	LOCAL CONST Robtarget Tr_meulage_bavure_P139 :=[[-127.011234375,174.2020625,18.5],[0.190442175287024,-0.303310117531916,0.790723364420333,-0.496478913383551],[0,0,0,0],[8.999999E+09,8.999999E+09,8.999999E+09,8.999999E+09,8.999999E+09,8.999999E+09]];
	LOCAL CONST Robtarget Tr_meulage_bavure_P140 :=[[-124.162203125,176.750703125,18.5],[0.192518086359884,-0.306201340616146,0.789260106907647,-0.496231809816071],[0,0,0,0],[8.999999E+09,8.999999E+09,8.999999E+09,8.999999E+09,8.999999E+09,8.999999E+09]];
	LOCAL CONST Robtarget Tr_meulage_bavure_P141 :=[[-122.8513828125,177.964453125,18.5],[0.194663155240253,-0.309123590669608,0.787712135243574,-0.49604279419567],[0,0,0,0],[8.999999E+09,8.999999E+09,8.999999E+09,8.999999E+09,8.999999E+09,8.999999E+09]];
	LOCAL CONST Robtarget Tr_meulage_bavure_P142 :=[[-119.9177578125,180.693,18.5],[0.196899901424474,-0.312103049014616,0.786062139961331,-0.495911713648938],[0,0,0,0],[8.999999E+09,8.999999E+09,8.999999E+09,8.999999E+09,8.999999E+09,8.999999E+09]];
	LOCAL CONST Robtarget Tr_meulage_bavure_P143 :=[[-116.7352265625,183.69171875,18.5],[0.199318008553782,-0.315263950024278,0.784246523173782,-0.49582089928832],[0,0,0,0],[8.999999E+09,8.999999E+09,8.999999E+09,8.999999E+09,8.999999E+09,8.999999E+09]];
	LOCAL CONST Robtarget Tr_meulage_bavure_P144 :=[[-116.454375,183.9246875,18.5],[0.20211682598174,-0.318902881092808,0.782129693912803,-0.495704431073234],[0,0,0,0],[8.999999E+09,8.999999E+09,8.999999E+09,8.999999E+09,8.999999E+09,8.999999E+09]];
	LOCAL CONST Robtarget Tr_meulage_bavure_P145 :=[[-112.0714453125,188.2565625,18.5],[0.205596230982278,-0.323472429632436,0.779505217686998,-0.495446659765022],[0,0,0,0],[8.999999E+09,8.999999E+09,8.999999E+09,8.999999E+09,8.999999E+09,8.999999E+09]];
	LOCAL CONST Robtarget Tr_meulage_bavure_P146 :=[[-110.354734375,189.926171875,18.5],[0.210070493146241,-0.329436360615377,0.776142089251371,-0.494919720264112],[0,0,0,0],[8.999999E+09,8.999999E+09,8.999999E+09,8.999999E+09,8.999999E+09,8.999999E+09]];
	LOCAL CONST Robtarget Tr_meulage_bavure_P147 :=[[-106.4182109375,193.63390625,18.5],[0.215682425483319,-0.33696654676811,0.771899664135642,-0.494070385880484],[0,0,0,0],[8.999999E+09,8.999999E+09,8.999999E+09,8.999999E+09,8.999999E+09,8.999999E+09]];
	LOCAL CONST Robtarget Tr_meulage_bavure_P148 :=[[-103.6989765625,196.126,18.5],[0.222270904527529,-0.345759095574698,0.766835763229423,-0.492959638368325],[0,0,0,0],[8.999999E+09,8.999999E+09,8.999999E+09,8.999999E+09,8.999999E+09,8.999999E+09]];
	LOCAL CONST Robtarget Tr_meulage_bavure_P149 :=[[-101.426390625,198.445984375,18.5],[0.229322634138018,-0.354960138136149,0.761267985475532,-0.491818547938559],[0,0,0,0],[8.999999E+09,8.999999E+09,8.999999E+09,8.999999E+09,8.999999E+09,8.999999E+09]];
	LOCAL CONST Robtarget Tr_meulage_bavure_P150 :=[[-101.17571875,198.708734375,18.5],[0.236006383142285,-0.363228319091028,0.755788103274612,-0.491070787437991],[0,0,0,0],[8.999999E+09,8.999999E+09,8.999999E+09,8.999999E+09,8.999999E+09,8.999999E+09]];
	LOCAL CONST Robtarget Tr_meulage_bavure_P151 :=[[-100.905703125,199.091640625,18.5],[0.241370828071747,-0.36906936863497,0.751137903082245,-0.491243091599823],[0,0,0,0],[8.999999E+09,8.999999E+09,8.999999E+09,8.999999E+09,8.999999E+09,8.999999E+09]];
	LOCAL CONST Robtarget Tr_meulage_bavure_P152 :=[[-99.122953125,201.35684375,18.5],[0.244403323371577,-0.370940628519687,0.748128933610927,-0.492923081557889],[0,0,0,0],[8.999999E+09,8.999999E+09,8.999999E+09,8.999999E+09,8.999999E+09,8.999999E+09]];
	LOCAL CONST Robtarget Tr_meulage_bavure_P153 :=[[-96.8828125,205.6408125,18.5],[0.244018753605267,-0.367253165730394,0.747565690475479,-0.496714705413334],[0,0,0,0],[8.999999E+09,8.999999E+09,8.999999E+09,8.999999E+09,8.999999E+09,8.999999E+09]];
	LOCAL CONST Robtarget Tr_meulage_bavure_P154 :=[[-96.362,206.638734375,18.5],[0.239111744899531,-0.356478263353551,0.750077508931146,-0.50312279992382],[0,0,0,0],[8.999999E+09,8.999999E+09,8.999999E+09,8.999999E+09,8.999999E+09,8.999999E+09]];
	LOCAL CONST Robtarget Tr_meulage_bavure_P155 :=[[-95.8127421875,207.699921875,18.5],[0.228678070464608,-0.337329813828571,0.755875580230949,-0.512412962366772],[0,0,0,0],[8.999999E+09,8.999999E+09,8.999999E+09,8.999999E+09,8.999999E+09,8.999999E+09]];
	LOCAL CONST Robtarget Tr_meulage_bavure_P156 :=[[-94.308015625,209.90903125,18.5],[0.212075421526648,-0.309184782305918,0.764495371744153,-0.524381171054517],[0,0,0,0],[8.999999E+09,8.999999E+09,8.999999E+09,8.999999E+09,8.999999E+09,8.999999E+09]];
	LOCAL CONST Robtarget Tr_meulage_bavure_P157 :=[[-93.75003125,210.7380625,18.5],[0.189378915500843,-0.272552593388089,0.774672329708009,-0.538268977172116],[0,0,0,0],[8.999999E+09,8.999999E+09,8.999999E+09,8.999999E+09,8.999999E+09,8.999999E+09]];
	LOCAL CONST Robtarget Tr_meulage_bavure_P158 :=[[-91.9986875,212.56409375,18.5],[0.161390602222789,-0.22902506301056,0.784689128838321,-0.552958918103443],[0,0,0,0],[8.999999E+09,8.999999E+09,8.999999E+09,8.999999E+09,8.999999E+09,8.999999E+09]];
	LOCAL CONST Robtarget Tr_meulage_bavure_P159 :=[[-91.4162265625,213.00103125,18.5],[0.129000654455637,-0.180301065959294,0.793038362347405,-0.567398019567663],[0,0,0,0],[8.999999E+09,8.999999E+09,8.999999E+09,8.999999E+09,8.999999E+09,8.999999E+09]];
	LOCAL CONST Robtarget Tr_meulage_bavure_P160 :=[[-91.3440546875,213.013484375,18.5],[0.0922817945694316,-0.126902080153844,0.798750290191089,-0.580842410954403],[0,0,0,0],[8.999999E+09,8.999999E+09,8.999999E+09,8.999999E+09,8.999999E+09,8.999999E+09]];
	LOCAL CONST Robtarget Tr_meulage_bavure_P161 :=[[-89.162078125,213.66828125,18.5],[0.0503174553587556,-0.0680160169269533,0.801040840932036,-0.592600663420577],[0,0,0,0],[8.999999E+09,8.999999E+09,8.999999E+09,8.999999E+09,8.999999E+09,8.999999E+09]];
	LOCAL CONST Robtarget Tr_meulage_bavure_P162 :=[[-88.3440546875,213.92571875,18.5],[0.00252406567631668,-0.00335106739002913,0.798759606326067,-0.601635679412081],[0,0,0,0],[8.999999E+09,8.999999E+09,8.999999E+09,8.999999E+09,8.999999E+09,8.999999E+09]];
	LOCAL CONST Robtarget Tr_meulage_bavure_P163 :=[[-87.4652109375,213.682671875,18.5],[0.0493797498258951,-0.0643494973435124,-0.79072352084382,0.606775985090975],[0,0,0,0],[8.999999E+09,8.999999E+09,8.999999E+09,8.999999E+09,8.999999E+09,8.999999E+09]];
	LOCAL CONST Robtarget Tr_meulage_bavure_P164 :=[[-85.52471875,212.9560625,18.5],[0.100577948139047,-0.128593194746078,-0.777116334377217,0.607814173458676],[0,0,0,0],[8.999999E+09,8.999999E+09,8.999999E+09,8.999999E+09,8.999999E+09,8.999999E+09]];
	LOCAL CONST Robtarget Tr_meulage_bavure_P165 :=[[-84.909671875,212.780703125,18.5],[0.145497398822093,-0.182465256610375,-0.760270957778014,0.606238408404991],[0,0,0,0],[8.999999E+09,8.999999E+09,8.999999E+09,8.999999E+09,8.999999E+09,8.999999E+09]];
	LOCAL CONST Robtarget Tr_meulage_bavure_P166 :=[[-84.38684375,212.302609375,18.5],[0.1809439145775,-0.222567903189488,-0.743324803089797,0.604310404807596],[0,0,0,0],[8.999999E+09,8.999999E+09,8.999999E+09,8.999999E+09,8.999999E+09,8.999999E+09]];
	LOCAL CONST Robtarget Tr_meulage_bavure_P167 :=[[-83.17071875,211.42740625,18.5],[0.206769871621223,-0.249506095485494,-0.728419709809437,0.603653588464826],[0,0,0,0],[8.999999E+09,8.999999E+09,8.999999E+09,8.999999E+09,8.999999E+09,8.999999E+09]];
	LOCAL CONST Robtarget Tr_meulage_bavure_P168 :=[[-80.6744375,209.227359375,18.5],[0.2245846611902,-0.265959685221285,-0.716250493467956,0.604824277292163],[0,0,0,0],[8.999999E+09,8.999999E+09,8.999999E+09,8.999999E+09,8.999999E+09,8.999999E+09]];
	LOCAL CONST Robtarget Tr_meulage_bavure_P169 :=[[-78.3284921875,206.867765625,18.5],[0.236502082156785,-0.27502158665567,-0.706570578623321,0.607608352010412],[0,0,0,0],[8.999999E+09,8.999999E+09,8.999999E+09,8.999999E+09,8.999999E+09,8.999999E+09]];
	LOCAL CONST Robtarget Tr_meulage_bavure_P170 :=[[-78.2308046875,206.771265625,18.5],[0.244452716764455,-0.279349107845849,-0.698778256751739,0.611486625449164],[0,0,0,0],[8.999999E+09,8.999999E+09,8.999999E+09,8.999999E+09,8.999999E+09,8.999999E+09]];
	LOCAL CONST Robtarget Tr_meulage_bavure_P171 :=[[-78.2126171875,206.752984375,18.5],[0.249940631640984,-0.280932693864888,-0.692284568560228,0.61591280089482],[0,0,0,0],[8.999999E+09,8.999999E+09,8.999999E+09,8.999999E+09,8.999999E+09,8.999999E+09]];
	LOCAL CONST Robtarget Tr_meulage_bavure_P172 :=[[-78.1261015625,206.67025,18.5],[0.253945556991537,-0.28103631183058,-0.686678755595343,0.620485722745459],[0,0,0,0],[8.999999E+09,8.999999E+09,8.999999E+09,8.999999E+09,8.999999E+09,8.999999E+09]];
	LOCAL CONST Robtarget Tr_meulage_bavure_P173 :=[[-71.4190078125,200.202265625,18.5],[0.256989223430704,-0.28033188921564,-0.681743993140734,0.62497655855704],[0,0,0,0],[8.999999E+09,8.999999E+09,8.999999E+09,8.999999E+09,8.999999E+09,8.999999E+09]];
	LOCAL CONST Robtarget Tr_meulage_bavure_P174 :=[[-69.085453125,198.020046875,18.5],[0.259270883175515,-0.279099527691383,-0.677410081478571,0.629283437165663],[0,0,0,0],[8.999999E+09,8.999999E+09,8.999999E+09,8.999999E+09,8.999999E+09,8.999999E+09]];
	LOCAL CONST Robtarget Tr_meulage_bavure_P175 :=[[-67.2452734375,196.310515625,18.5],[0.260735300009118,-0.277312443707638,-0.673704973181902,0.633432333405887],[0,0,0,0],[8.999999E+09,8.999999E+09,8.999999E+09,8.999999E+09,8.999999E+09,8.999999E+09]];
	LOCAL CONST Robtarget Tr_meulage_bavure_P176 :=[[-65.573640625,194.69784375,18.5],[0.261286645683991,-0.274898585018902,-0.670672090802852,0.63746294273467],[0,0,0,0],[8.999999E+09,8.999999E+09,8.999999E+09,8.999999E+09,8.999999E+09,8.999999E+09]];
	LOCAL CONST Robtarget Tr_meulage_bavure_P177 :=[[-61.1885078125,190.282375,18.5],[0.260938532941136,-0.27189092460859,-0.668297686772354,0.641377119171501],[0,0,0,0],[8.999999E+09,8.999999E+09,8.999999E+09,8.999999E+09,8.999999E+09,8.999999E+09]];
	LOCAL CONST Robtarget Tr_meulage_bavure_P178 :=[[-60.0119609375,189.182125,18.5],[0.259877003328182,-0.268486303796629,-0.666487105011264,0.645115483203196],[0,0,0,0],[8.999999E+09,8.999999E+09,8.999999E+09,8.999999E+09,8.999999E+09,8.999999E+09]];
	LOCAL CONST Robtarget Tr_meulage_bavure_P179 :=[[-56.05679296875,185.29428125,18.5],[0.258463269105114,-0.265048735721945,-0.665076369193805,0.648551716793412],[0,0,0,0],[8.999999E+09,8.999999E+09,8.999999E+09,8.999999E+09,8.999999E+09,8.999999E+09]];
	LOCAL CONST Robtarget Tr_meulage_bavure_P180 :=[[-54.05676171875,183.442875,18.5],[0.257127057998321,-0.26199711676235,-0.663881001079455,0.651540638225341],[0,0,0,0],[8.999999E+09,8.999999E+09,8.999999E+09,8.999999E+09,8.999999E+09,8.999999E+09]];
	LOCAL CONST Robtarget Tr_meulage_bavure_P181 :=[[-52.6292734375,182.20425,18.5],[0.25621924205441,-0.259657247241297,-0.662753509176958,0.653978287124094],[0,0,0,0],[8.999999E+09,8.999999E+09,8.999999E+09,8.999999E+09,8.999999E+09,8.999999E+09]];
	LOCAL CONST Robtarget Tr_meulage_bavure_P182 :=[[-50.96499609375,180.630546875,18.5],[0.25590306679538,-0.258163340391161,-0.661625616240868,0.655832946730102],[0,0,0,0],[8.999999E+09,8.999999E+09,8.999999E+09,8.999999E+09,8.999999E+09,8.999999E+09]];
	LOCAL CONST Robtarget Tr_meulage_bavure_P183 :=[[-48.427734375,178.2460625,18.5],[0.256144256103112,-0.257446199530212,-0.66049710199585,0.657156870669339],[0,0,0,0],[8.999999E+09,8.999999E+09,8.999999E+09,8.999999E+09,8.999999E+09,8.999999E+09]];
	LOCAL CONST Robtarget Tr_meulage_bavure_P184 :=[[-43.8993828125,173.85284375,18.5],[0.25677948279759,-0.257318314364314,-0.659420499348961,0.658039654842531],[0,0,0,0],[8.999999E+09,8.999999E+09,8.999999E+09,8.999999E+09,8.999999E+09,8.999999E+09]];
	LOCAL CONST Robtarget Tr_meulage_bavure_P185 :=[[-43.0797734375,173.100734375,18.5],[0.257617067745429,-0.257566704531451,-0.658453973298864,0.658582723862382],[0,0,0,0],[8.999999E+09,8.999999E+09,8.999999E+09,8.999999E+09,8.999999E+09,8.999999E+09]];
	LOCAL CONST Robtarget Tr_meulage_bavure_P186 :=[[-41.48028515625,171.667078125,18.5],[0.258515279559301,-0.258032413744623,-0.657635522171516,0.658866180396063],[0,0,0,0],[8.999999E+09,8.999999E+09,8.999999E+09,8.999999E+09,8.999999E+09,8.999999E+09]];
	LOCAL CONST Robtarget Tr_meulage_bavure_P187 :=[[-39.0978984375,169.191015625,18.5],[0.259401397972076,-0.258624835211619,-0.656973453033344,0.658946121736322],[0,0,0,0],[8.999999E+09,8.999999E+09,8.999999E+09,8.999999E+09,8.999999E+09,8.999999E+09]];
	LOCAL CONST Robtarget Tr_meulage_bavure_P188 :=[[-38.23126171875,168.3086875,18.5],[0.260254131673374,-0.259304274264351,-0.656454947464892,0.658859607385399],[0,0,0,0],[8.999999E+09,8.999999E+09,8.999999E+09,8.999999E+09,8.999999E+09,8.999999E+09]];
	LOCAL CONST Robtarget Tr_meulage_bavure_P189 :=[[-35.4189765625,165.67340625,18.5],[0.26105089862492,-0.260039320067026,-0.656077957241587,0.658630165091083],[0,0,0,0],[8.999999E+09,8.999999E+09,8.999999E+09,8.999999E+09,8.999999E+09,8.999999E+09]];
	LOCAL CONST Robtarget Tr_meulage_bavure_P190 :=[[-34.5329296875,164.8164375,18.5],[0.261759260875739,-0.2607857252386,-0.655841250825685,0.65828956286194],[0,0,0,0],[8.999999E+09,8.999999E+09,8.999999E+09,8.999999E+09,8.999999E+09,8.999999E+09]];
	LOCAL CONST Robtarget Tr_meulage_bavure_P191 :=[[-31.362640625,161.758390625,18.5],[0.262331145993118,-0.261476154519974,-0.655742298154861,0.657886486310493],[0,0,0,0],[8.999999E+09,8.999999E+09,8.999999E+09,8.999999E+09,8.999999E+09,8.999999E+09]];
	LOCAL CONST Robtarget Tr_meulage_bavure_P192 :=[[-30.35272265625,160.788,18.5],[0.262709953836354,-0.262042168547561,-0.655790615320609,0.657461824683083],[0,0,0,0],[8.999999E+09,8.999999E+09,8.999999E+09,8.999999E+09,8.999999E+09,8.999999E+09]];
	LOCAL CONST Robtarget Tr_meulage_bavure_P193 :=[[-30.05163671875,160.490046875,18.5],[0.262861381702475,-0.262436848617029,-0.655986833448376,0.657047995841857],[0,0,0,0],[8.999999E+09,8.999999E+09,8.999999E+09,8.999999E+09,8.999999E+09,8.999999E+09]];
	LOCAL CONST Robtarget Tr_meulage_bavure_P194 :=[[-28.3164375,158.80840625,18.5],[0.262783789530265,-0.262648406055636,-0.656321684574613,0.656659988969703],[0,0,0,0],[8.999999E+09,8.999999E+09,8.999999E+09,8.999999E+09,8.999999E+09,8.999999E+09]];
	LOCAL CONST Robtarget Tr_meulage_bavure_P195 :=[[-23.402556640625,154.107609375,18.5],[0.262525712244518,-0.262712755695221,-0.6567633663921,0.656295770953042],[0,0,0,0],[8.999999E+09,8.999999E+09,8.999999E+09,8.999999E+09,8.999999E+09,8.999999E+09]];
	LOCAL CONST Robtarget Tr_meulage_bavure_P196 :=[[-20.412109375,151.27234375,18.5],[0.262165502805967,-0.262695654197738,-0.657267884152523,0.655941438594775],[0,0,0,0],[8.999999E+09,8.999999E+09,8.999999E+09,8.999999E+09,8.999999E+09,8.999999E+09]];
	LOCAL CONST Robtarget Tr_meulage_bavure_P197 :=[[-16.22085546875,147.224703125,18.5],[0.261778886975614,-0.262664639311416,-0.657796488234147,0.655578280341895],[0,0,0,0],[8.999999E+09,8.999999E+09,8.999999E+09,8.999999E+09,8.999999E+09,8.999999E+09]];
	LOCAL CONST Robtarget Tr_meulage_bavure_P198 :=[[-14.92822265625,146.00884375,18.5],[0.261413667950097,-0.262658057795985,-0.658319979987044,0.655201070537568],[0,0,0,0],[8.999999E+09,8.999999E+09,8.999999E+09,8.999999E+09,8.999999E+09,8.999999E+09]];
	LOCAL CONST Robtarget Tr_meulage_bavure_P199 :=[[-11.3293759765625,142.66771875,18.5],[0.261077038101035,-0.262673384522033,-0.658825150616152,0.654821268863295],[0,0,0,0],[8.999999E+09,8.999999E+09,8.999999E+09,8.999999E+09,8.999999E+09,8.999999E+09]];
	LOCAL CONST Robtarget Tr_meulage_bavure_P200 :=[[-6.89715576171875,138.38053125,18.5],[0.260745670082175,-0.262685448847026,-0.659319494058335,0.654450804302429],[0,0,0,0],[8.999999E+09,8.999999E+09,8.999999E+09,8.999999E+09,8.999999E+09,8.999999E+09]];
	LOCAL CONST Robtarget Tr_meulage_bavure_P201 :=[[-5.350982421875,136.87134375,18.5],[0.260409251060274,-0.262675169776875,-0.659798086716118,0.654106460685619],[0,0,0,0],[8.999999E+09,8.999999E+09,8.999999E+09,8.999999E+09,8.999999E+09,8.999999E+09]];
	LOCAL CONST Robtarget Tr_meulage_bavure_P202 :=[[-2.4296875,134.151703125,18.5],[0.260088169520179,-0.262658023455088,-0.660247459881271,0.653787579042795],[0,0,0,0],[8.999999E+09,8.999999E+09,8.999999E+09,8.999999E+09,8.999999E+09,8.999999E+09]];
	LOCAL CONST Robtarget Tr_meulage_bavure_P203 :=[[0.08966064453125,131.796015625,18.5],[0.259835082530743,-0.2626829624302,-0.660641959735919,0.653479603485389],[0,0,0,0],[8.999999E+09,8.999999E+09,8.999999E+09,8.999999E+09,8.999999E+09,8.999999E+09]];
	LOCAL CONST Robtarget Tr_meulage_bavure_P204 :=[[10.1913759765625,122.3306875,18.5],[0.259705705094535,-0.262804592862917,-0.660957113707128,0.653163368960209],[0,0,0,0],[8.999999E+09,8.999999E+09,8.999999E+09,8.999999E+09,8.999999E+09,8.999999E+09]];
	LOCAL CONST Robtarget Tr_meulage_bavure_P205 :=[[11.085693359375,121.4689921875,18.5],[0.259721319569318,-0.263044848045246,-0.661184340698121,0.652830385087595],[0,0,0,0],[8.999999E+09,8.999999E+09,8.999999E+09,8.999999E+09,8.999999E+09,8.999999E+09]];
	LOCAL CONST Robtarget Tr_meulage_bavure_P206 :=[[17.055603515625,115.9521796875,18.5],[0.259852146003557,-0.263371187191271,-0.661332752660767,0.652496337332969],[0,0,0,0],[8.999999E+09,8.999999E+09,8.999999E+09,8.999999E+09,8.999999E+09,8.999999E+09]];
	LOCAL CONST Robtarget Tr_meulage_bavure_P207 :=[[21.760802734375,111.515078125,18.5],[0.260013158425684,-0.263699039363099,-0.661438173618062,0.652192852280122],[0,0,0,0],[8.999999E+09,8.999999E+09,8.999999E+09,8.999999E+09,8.999999E+09,8.999999E+09]];
	LOCAL CONST Robtarget Tr_meulage_bavure_P208 :=[[27.258392578125,106.207,18.5],[0.260100750372149,-0.263922045498253,-0.661541379549992,0.651963002553792],[0,0,0,0],[8.999999E+09,8.999999E+09,8.999999E+09,8.999999E+09,8.999999E+09,8.999999E+09]];
	LOCAL CONST Robtarget Tr_meulage_bavure_P209 :=[[28.722015625,104.805484375,18.5],[0.260029172084293,-0.263956096433542,-0.661680511567474,0.651836566504618],[0,0,0,0],[8.999999E+09,8.999999E+09,8.999999E+09,8.999999E+09,8.999999E+09,8.999999E+09]];
	LOCAL CONST Robtarget Tr_meulage_bavure_P210 :=[[29.41101171875,104.1642734375,18.5],[0.259754440439883,-0.263762334346421,-0.661879667905148,0.651822343024279],[0,0,0,0],[8.999999E+09,8.999999E+09,8.999999E+09,8.999999E+09,8.999999E+09,8.999999E+09]];
	LOCAL CONST Robtarget Tr_meulage_bavure_P211 :=[[32.655669921875,101.1337265625,18.5],[0.259303936814273,-0.263365032759278,-0.662124089734479,0.651914118320513],[0,0,0,0],[8.999999E+09,8.999999E+09,8.999999E+09,8.999999E+09,8.999999E+09,8.999999E+09]];
	LOCAL CONST Robtarget Tr_meulage_bavure_P212 :=[[33.78524609375,100.0587734375,18.5],[0.258758312179959,-0.262849754312713,-0.662384650536248,0.65207416546701],[0,0,0,0],[8.999999E+09,8.999999E+09,8.999999E+09,8.999999E+09,8.999999E+09,8.999999E+09]];
	LOCAL CONST Robtarget Tr_meulage_bavure_P213 :=[[36.34820703125,97.613921875,18.5],[0.258230341869406,-0.262336593473032,-0.662621353895246,0.652249602242122],[0,0,0,0],[8.999999E+09,8.999999E+09,8.999999E+09,8.999999E+09,8.999999E+09,8.999999E+09]];
	LOCAL CONST Robtarget Tr_meulage_bavure_P214 :=[[36.68661328125,97.301265625,18.5],[0.257838264135803,-0.261942230185288,-0.662783034784466,0.652398916610755],[0,0,0,0],[8.999999E+09,8.999999E+09,8.999999E+09,8.999999E+09,8.999999E+09,8.999999E+09]];
	LOCAL CONST Robtarget Tr_meulage_bavure_P215 :=[[41.70132421875,92.63553125,18.5],[0.257661233706871,-0.261751929505443,-0.662843156043849,0.652484150405709],[0,0,0,0],[8.999999E+09,8.999999E+09,8.999999E+09,8.999999E+09,8.999999E+09,8.999999E+09]];
	LOCAL CONST Robtarget Tr_meulage_bavure_P216 :=[[42.19903515625,92.1639375,18.5],[0.257726518582814,-0.26179495027106,-0.662792605179694,0.652492458309572],[0,0,0,0],[8.999999E+09,8.999999E+09,8.999999E+09,8.999999E+09,8.999999E+09,8.999999E+09]];
	LOCAL CONST Robtarget Tr_meulage_bavure_P217 :=[[46.81198046875,87.720828125,18.5],[0.257999907114851,-0.262035769496674,-0.662644346135569,0.65243832962785],[0,0,0,0],[8.999999E+09,8.999999E+09,8.999999E+09,8.999999E+09,8.999999E+09,8.999999E+09]];
	LOCAL CONST Robtarget Tr_meulage_bavure_P218 :=[[49.733125,84.880984375,18.5],[0.25840165568085,-0.262392247290674,-0.662429146914292,0.652354595462888],[0,0,0,0],[8.999999E+09,8.999999E+09,8.999999E+09,8.999999E+09,8.999999E+09,8.999999E+09]];
	LOCAL CONST Robtarget Tr_meulage_bavure_P219 :=[[53.43625,81.315796875,18.5],[0.258834760496953,-0.262763022767383,-0.662183038441192,0.652283515218209],[0,0,0,0],[8.999999E+09,8.999999E+09,8.999999E+09,8.999999E+09,8.999999E+09,8.999999E+09]];
	LOCAL CONST Robtarget Tr_meulage_bavure_P220 :=[[53.95355078125,80.838375,18.5],[0.259211162458601,-0.263064591543837,-0.661947709033417,0.652251350660269],[0,0,0,0],[8.999999E+09,8.999999E+09,8.999999E+09,8.999999E+09,8.999999E+09,8.999999E+09]];
	LOCAL CONST Robtarget Tr_meulage_bavure_P221 :=[[54.826875,80.0061015625,18.5],[0.259488029803717,-0.263250179274638,-0.661737089246687,0.652280101042319],[0,0,0,0],[8.999999E+09,8.999999E+09,8.999999E+09,8.999999E+09,8.999999E+09,8.999999E+09]];
	LOCAL CONST Robtarget Tr_meulage_bavure_P222 :=[[60.5829453125,74.60928125,18.5],[0.259674946248655,-0.26332359323042,-0.661541189697748,0.65237478635541],[0,0,0,0],[8.999999E+09,8.999999E+09,8.999999E+09,8.999999E+09,8.999999E+09,8.999999E+09]];
	LOCAL CONST Robtarget Tr_meulage_bavure_P223 :=[[63.79837109375,71.542265625,18.5],[0.259811135200041,-0.263327157504758,-0.661346749701084,0.652516251756492],[0,0,0,0],[8.999999E+09,8.999999E+09,8.999999E+09,8.999999E+09,8.999999E+09,8.999999E+09]];
	LOCAL CONST Robtarget Tr_meulage_bavure_P224 :=[[64.75128125,70.6356171875,18.5],[0.259950506966493,-0.263316075940902,-0.661132529812424,0.652682278067033],[0,0,0,0],[8.999999E+09,8.999999E+09,8.999999E+09,8.999999E+09,8.999999E+09,8.999999E+09]];
	LOCAL CONST Robtarget Tr_meulage_bavure_P225 :=[[65.2604375,70.1572890625,18.5],[0.260128633947986,-0.2633247332003,-0.660882480354013,0.65286103103683],[0,0,0,0],[8.999999E+09,8.999999E+09,8.999999E+09,8.999999E+09,8.999999E+09,8.999999E+09]];
	LOCAL CONST Robtarget Tr_meulage_bavure_P226 :=[[74.823515625,61.04348828125,18.5],[0.260357808457022,-0.263364331937732,-0.660590435750362,0.653049245029497],[0,0,0,0],[8.999999E+09,8.999999E+09,8.999999E+09,8.999999E+09,8.999999E+09,8.999999E+09]];
	LOCAL CONST Robtarget Tr_meulage_bavure_P227 :=[[74.958921875,60.909578125,18.5],[0.260635977982767,-0.263433479938855,-0.660258045133076,0.65324650972303],[0,0,0,0],[8.999999E+09,8.999999E+09,8.999999E+09,8.999999E+09,8.999999E+09,8.999999E+09]];
	LOCAL CONST Robtarget Tr_meulage_bavure_P228 :=[[75.2834765625,60.5998828125,18.5],[0.260959923728408,-0.263534304872991,-0.659892312110163,0.653446038155162],[0,0,0,0],[8.999999E+09,8.999999E+09,8.999999E+09,8.999999E+09,8.999999E+09,8.999999E+09]];
	LOCAL CONST Robtarget Tr_meulage_bavure_P229 :=[[76.818203125,59.1343984375,18.5],[0.261348507260307,-0.263684070418043,-0.65948391843562,0.653642585887258],[0,0,0,0],[8.999999E+09,8.999999E+09,8.999999E+09,8.999999E+09,8.999999E+09,8.999999E+09]];
	LOCAL CONST Robtarget Tr_meulage_bavure_P230 :=[[80.37746875,55.78567578125,18.5],[0.261818900977442,-0.263905367215071,-0.659031593273065,0.653821213569893],[0,0,0,0],[8.999999E+09,8.999999E+09,8.999999E+09,8.999999E+09,8.999999E+09,8.999999E+09]];
	LOCAL CONST Robtarget Tr_meulage_bavure_P231 :=[[82.7379765625,53.54480078125,18.5],[0.262374279281103,-0.264207097898495,-0.658540178166431,0.653971850106946],[0,0,0,0],[8.999999E+09,8.999999E+09,8.999999E+09,8.999999E+09,8.999999E+09,8.999999E+09]];
	LOCAL CONST Robtarget Tr_meulage_bavure_P232 :=[[85.722015625,50.74478125,18.5],[0.262980865779189,-0.264558020476555,-0.658026347051853,0.654103542737042],[0,0,0,0],[8.999999E+09,8.999999E+09,8.999999E+09,8.999999E+09,8.999999E+09,8.999999E+09]];
	LOCAL CONST Robtarget Tr_meulage_bavure_P233 :=[[86.495359375,50.05071875,18.5],[0.263564261369973,-0.264894657473782,-0.657531980936437,0.654229619182863],[0,0,0,0],[8.999999E+09,8.999999E+09,8.999999E+09,8.999999E+09,8.999999E+09,8.999999E+09]];
	LOCAL CONST Robtarget Tr_meulage_bavure_P234 :=[[91.53765625,45.121796875,18.5],[0.264038385192771,-0.265135745170548,-0.657097214729498,0.654377580737901],[0,0,0,0],[8.999999E+09,8.999999E+09,8.999999E+09,8.999999E+09,8.999999E+09,8.999999E+09]];
	LOCAL CONST Robtarget Tr_meulage_bavure_P235 :=[[91.7916875,44.872375,18.5],[0.264276966366081,-0.26516564492129,-0.656784358273732,0.654583205199141],[0,0,0,0],[8.999999E+09,8.999999E+09,8.999999E+09,8.999999E+09,8.999999E+09,8.999999E+09]];
	LOCAL CONST Robtarget Tr_meulage_bavure_P236 :=[[92.083890625,44.57428125,18.5],[0.264130741135658,-0.264845550566766,-0.656664403634689,0.654892088004743],[0,0,0,0],[8.999999E+09,8.999999E+09,8.999999E+09,8.999999E+09,8.999999E+09,8.999999E+09]];
	LOCAL CONST Robtarget Tr_meulage_bavure_P237 :=[[92.758484375,43.960203125,18.5],[0.2634323732283,-0.264013117641807,-0.656809046399305,0.655364276579365],[0,0,0,0],[8.999999E+09,8.999999E+09,8.999999E+09,8.999999E+09,8.999999E+09,8.999999E+09]];
	LOCAL CONST Robtarget Tr_meulage_bavure_P238 :=[[94.1454453125,42.5842578125,18.5],[0.26198643820928,-0.262486825874829,-0.657308711312959,0.656055661105572],[0,0,0,0],[8.999999E+09,8.999999E+09,8.999999E+09,8.999999E+09,8.999999E+09,8.999999E+09]];
	LOCAL CONST Robtarget Tr_meulage_bavure_P239 :=[[94.8658125,41.89669921875,18.5],[0.259703936587452,-0.260184198391892,-0.658200547887968,0.656985606378198],[0,0,0,0],[8.999999E+09,8.999999E+09,8.999999E+09,8.999999E+09,8.999999E+09,8.999999E+09]];
	LOCAL CONST Robtarget Tr_meulage_bavure_P240 :=[[95.11734375,41.6527109375,18.5],[0.256743431384074,-0.257267124340212,-0.65941827594038,0.658075964103435],[0,0,0,0],[8.999999E+09,8.999999E+09,8.999999E+09,8.999999E+09,8.999999E+09,8.999999E+09]];
	LOCAL CONST Robtarget Tr_meulage_bavure_P241 :=[[96.8580625,40.081359375,18.5],[0.253611692690041,-0.254249223689498,-0.660766718478608,0.659109843148463],[0,0,0,0],[8.999999E+09,8.999999E+09,8.999999E+09,8.999999E+09,8.999999E+09,8.999999E+09]];
	LOCAL CONST Robtarget Tr_meulage_bavure_P242 :=[[98.404234375,38.6039140625,18.5],[0.251102642755858,-0.251926378039458,-0.661944594264948,0.65978020353172],[0,0,0,0],[8.999999E+09,8.999999E+09,8.999999E+09,8.999999E+09,8.999999E+09,8.999999E+09]];
	LOCAL CONST Robtarget Tr_meulage_bavure_P243 :=[[98.859375,38.1670234375,18.5],[0.250014871661718,-0.251102998309306,-0.662660299561253,0.659788735561196],[0,0,0,0],[8.999999E+09,8.999999E+09,8.999999E+09,8.999999E+09,8.999999E+09,8.999999E+09]];
	LOCAL CONST Robtarget Tr_meulage_bavure_P244 :=[[99.3323046875,37.7099921875,18.5],[0.250805849511644,-0.252239352394942,-0.66274047424979,0.658974050130418],[0,0,0,0],[8.999999E+09,8.999999E+09,8.999999E+09,8.999999E+09,8.999999E+09,8.999999E+09]];
	LOCAL CONST Robtarget Tr_meulage_bavure_P245 :=[[103.6297578125,33.65280078125,18.5],[0.253310213160779,-0.255177218529122,-0.662235775265235,0.65739052397417],[0,0,0,0],[8.999999E+09,8.999999E+09,8.999999E+09,8.999999E+09,8.999999E+09,8.999999E+09]];
	LOCAL CONST Robtarget Tr_meulage_bavure_P246 :=[[104.81625,32.4886484375,18.5],[0.25677611929244,-0.25916604636247,-0.661411386214233,0.655312111257016],[0,0,0,0],[8.999999E+09,8.999999E+09,8.999999E+09,8.999999E+09,8.999999E+09,8.999999E+09]];
	LOCAL CONST Robtarget Tr_meulage_bavure_P247 :=[[105.6639375,31.622771484375,18.5],[0.260206650483068,-0.263195321942458,-0.660634637752421,0.653132909103282],[0,0,0,0],[8.999999E+09,8.999999E+09,8.999999E+09,8.999999E+09,8.999999E+09,8.999999E+09]];
	LOCAL CONST Robtarget Tr_meulage_bavure_P248 :=[[106.382265625,31.046234375,18.5],[0.262750855464765,-0.266393885985042,-0.660241413100884,0.651212378482527],[0,0,0,0],[8.999999E+09,8.999999E+09,8.999999E+09,8.999999E+09,8.999999E+09,8.999999E+09]];
	LOCAL CONST Robtarget Tr_meulage_bavure_P249 :=[[107.8891015625,29.551390625,18.5],[0.263982593952903,-0.268315834441988,-0.660414033699996,0.649748495319301],[0,0,0,0],[8.999999E+09,8.999999E+09,8.999999E+09,8.999999E+09,8.999999E+09,8.999999E+09]];
	LOCAL CONST Robtarget Tr_meulage_bavure_P250 :=[[108.62771875,28.843537109375,18.5],[0.263952893247615,-0.268988684801326,-0.661130315255106,0.648753160952414],[0,0,0,0],[8.999999E+09,8.999999E+09,8.999999E+09,8.999999E+09,8.999999E+09,8.999999E+09]];
	LOCAL CONST Robtarget Tr_meulage_bavure_P251 :=[[112.0958828125,25.593505859375,18.5],[0.263037601677577,-0.268771657058905,-0.662225572151647,0.648097452590227],[0,0,0,0],[8.999999E+09,8.999999E+09,8.999999E+09,8.999999E+09,8.999999E+09,8.999999E+09]];
	LOCAL CONST Robtarget Tr_meulage_bavure_P252 :=[[117.3396640625,20.51574609375,18.5],[0.26172937870922,-0.268144924993792,-0.663478862004478,0.647604687439647],[0,0,0,0],[8.999999E+09,8.999999E+09,8.999999E+09,8.999999E+09,8.999999E+09,8.999999E+09]];
	LOCAL CONST Robtarget Tr_meulage_bavure_P253 :=[[117.563171875,20.302794921875,18.5],[0.26043211435292,-0.26750871992158,-0.6647110958406,0.647127002717375],[0,0,0,0],[8.999999E+09,8.999999E+09,8.999999E+09,8.999999E+09,8.999999E+09,8.999999E+09]];
	LOCAL CONST Robtarget Tr_meulage_bavure_P254 :=[[117.6695546875,20.203033203125,18.5],[0.259412524202119,-0.267117643872184,-0.665791857851134,0.646586814463761],[0,0,0,0],[8.999999E+09,8.999999E+09,8.999999E+09,8.999999E+09,8.999999E+09,8.999999E+09]];
	LOCAL CONST Robtarget Tr_meulage_bavure_P255 :=[[117.8055390625,20.072998046875,18.5],[0.258779385619435,-0.267066734528231,-0.666656937681159,0.645969903577894],[0,0,0,0],[8.999999E+09,8.999999E+09,8.999999E+09,8.999999E+09,8.999999E+09,8.999999E+09]];
	LOCAL CONST Robtarget Tr_meulage_bavure_P256 :=[[118.1591171875,19.7444765625,18.5],[0.258477945816715,-0.267295169833574,-0.667321956843276,0.645309111685921],[0,0,0,0],[8.999999E+09,8.999999E+09,8.999999E+09,8.999999E+09,8.999999E+09,8.999999E+09]];
	LOCAL CONST Robtarget Tr_meulage_bavure_P257 :=[[121.810484375,16.36737109375,18.5],[0.258382394356594,-0.267663963941661,-0.667828215829711,0.644670469957556],[0,0,0,0],[8.999999E+09,8.999999E+09,8.999999E+09,8.999999E+09,8.999999E+09,8.999999E+09]];
	LOCAL CONST Robtarget Tr_meulage_bavure_P258 :=[[124.4450703125,13.93145703125,18.5],[0.258330668513948,-0.267987374932702,-0.668224704779796,0.6441457727128],[0,0,0,0],[8.999999E+09,8.999999E+09,8.999999E+09,8.999999E+09,8.999999E+09,8.999999E+09]];
	LOCAL CONST Robtarget Tr_meulage_bavure_P259 :=[[126.9319453125,11.502837890625,18.5],[0.258162255629655,-0.268089090848659,-0.668569238233849,0.643813375772482],[0,0,0,0],[8.999999E+09,8.999999E+09,8.999999E+09,8.999999E+09,8.999999E+09,8.999999E+09]];
	LOCAL CONST Robtarget Tr_meulage_bavure_P260 :=[[128.69025,9.8183896484375,18.5],[0.257780134202139,-0.26786455633663,-0.668899383569445,0.643717015877105],[0,0,0,0],[8.999999E+09,8.999999E+09,8.999999E+09,8.999999E+09,8.999999E+09,8.999999E+09]];
	LOCAL CONST Robtarget Tr_meulage_bavure_P261 :=[[132.04846875,6.68276953125,18.5],[0.257188457009479,-0.267317027428435,-0.66921230787111,0.643856033148507],[0,0,0,0],[8.999999E+09,8.999999E+09,8.999999E+09,8.999999E+09,8.999999E+09,8.999999E+09]];
	LOCAL CONST Robtarget Tr_meulage_bavure_P262 :=[[133.398015625,5.3205869140625,18.5],[0.256525337159777,-0.266581023841979,-0.6694404245491,0.644188502770692],[0,0,0,0],[8.999999E+09,8.999999E+09,8.999999E+09,8.999999E+09,8.999999E+09,8.999999E+09]];
	LOCAL CONST Robtarget Tr_meulage_bavure_P263 :=[[134.411921875,4.41253662109375,18.5],[0.256028392471401,-0.265905990693878,-0.669486526635195,0.644617139871071],[0,0,0,0],[8.999999E+09,8.999999E+09,8.999999E+09,8.999999E+09,8.999999E+09,8.999999E+09]];
	LOCAL CONST Robtarget Tr_meulage_bavure_P264 :=[[139.8126875,-0.7569580078125,18.5],[0.255961038509432,-0.265567966011388,-0.669244427311966,0.645034494198277],[0,0,0,0],[8.999999E+09,8.999999E+09,8.999999E+09,8.999999E+09,8.999999E+09,8.999999E+09]];
	LOCAL CONST Robtarget Tr_meulage_bavure_P265 :=[[141.512578125,-2.3416748046875,18.5],[0.256502648532083,-0.265753924385189,-0.668642908331438,0.645366488212686],[0,0,0,0],[8.999999E+09,8.999999E+09,8.999999E+09,8.999999E+09,8.999999E+09,8.999999E+09]];
	LOCAL CONST Robtarget Tr_meulage_bavure_P266 :=[[142.39690625,-3.21923828125,18.5],[0.257645906569791,-0.266457293833768,-0.667688605001759,0.645609033503575],[0,0,0,0],[8.999999E+09,8.999999E+09,8.999999E+09,8.999999E+09,8.999999E+09,8.999999E+09]];
	LOCAL CONST Robtarget Tr_meulage_bavure_P267 :=[[144.952640625,-5.6247255859375,18.5],[0.259175691325742,-0.267460753452128,-0.666477971183888,0.645832656587798],[0,0,0,0],[8.999999E+09,8.999999E+09,8.999999E+09,8.999999E+09,8.999999E+09,8.999999E+09]];
	LOCAL CONST Robtarget Tr_meulage_bavure_P268 :=[[145.87896875,-6.51544189453125,18.5],[0.260740620240717,-0.268407635998818,-0.665164380016557,0.64616407935694],[0,0,0,0],[8.999999E+09,8.999999E+09,8.999999E+09,8.999999E+09,8.999999E+09,8.999999E+09]];
	LOCAL CONST Robtarget Tr_meulage_bavure_P269 :=[[147.8985625,-8.35919140625,18.5],[0.261983114518038,-0.268936860917328,-0.663903803180018,0.646737622742384],[0,0,0,0],[8.999999E+09,8.999999E+09,8.999999E+09,8.999999E+09,8.999999E+09,8.999999E+09]];
	LOCAL CONST Robtarget Tr_meulage_bavure_P270 :=[[148.7679375,-9.187408203125,18.5],[0.262677251096978,-0.268827508739435,-0.662798331235698,0.647634777025028],[0,0,0,0],[8.999999E+09,8.999999E+09,8.999999E+09,8.999999E+09,8.999999E+09,8.999999E+09]];
	LOCAL CONST Robtarget Tr_meulage_bavure_P271 :=[[152.97125,-13.264220703125,18.5],[0.262779930489003,-0.268053525089936,-0.661876788472569,0.648855247879134],[0,0,0,0],[8.999999E+09,8.999999E+09,8.999999E+09,8.999999E+09,8.999999E+09,8.999999E+09]];
	LOCAL CONST Robtarget Tr_meulage_bavure_P272 :=[[153.766046875,-14.0890810546875,18.5],[0.262417297149559,-0.266760691686163,-0.661094542801443,0.650330609002829],[0,0,0,0],[8.999999E+09,8.999999E+09,8.999999E+09,8.999999E+09,8.999999E+09,8.999999E+09]];
	LOCAL CONST Robtarget Tr_meulage_bavure_P273 :=[[154.1666875,-14.422607421875,18.5],[0.261801719711089,-0.265179245227982,-0.660370277161613,0.651959296657489],[0,0,0,0],[8.999999E+09,8.999999E+09,8.999999E+09,8.999999E+09,8.999999E+09,8.999999E+09]];
	LOCAL CONST Robtarget Tr_meulage_bavure_P274 :=[[157.0810625,-17.1715390625,18.5],[0.261137880333805,-0.263527206763498,-0.659626651937043,0.653646004198391],[0,0,0,0],[8.999999E+09,8.999999E+09,8.999999E+09,8.999999E+09,8.999999E+09,8.999999E+09]];
	LOCAL CONST Robtarget Tr_meulage_bavure_P275 :=[[158.70325,-18.534728515625,18.5],[0.260564095469008,-0.261958083629703,-0.658821485772524,0.6553156220158],[0,0,0,0],[8.999999E+09,8.999999E+09,8.999999E+09,8.999999E+09,8.999999E+09,8.999999E+09]];
	LOCAL CONST Robtarget Tr_meulage_bavure_P276 :=[[159.789921875,-19.60949609375,18.5],[0.260129835582888,-0.260540468392887,-0.657956933011838,0.656919939772641],[0,0,0,0],[8.999999E+09,8.999999E+09,8.999999E+09,8.999999E+09,8.999999E+09,8.999999E+09]];
	LOCAL CONST Robtarget Tr_meulage_bavure_P277 :=[[160.903265625,-20.70852734375,18.5],[0.259819170030927,-0.259261804049378,-0.657046088819179,0.658458619058876],[0,0,0,0],[8.999999E+09,8.999999E+09,8.999999E+09,8.999999E+09,8.999999E+09,8.999999E+09]];
	LOCAL CONST Robtarget Tr_meulage_bavure_P278 :=[[163.091734375,-22.7197578125,18.5],[0.259568059571996,-0.258070380720333,-0.656129873886991,0.659937640719131],[0,0,0,0],[8.999999E+09,8.999999E+09,8.999999E+09,8.999999E+09,8.999999E+09,8.999999E+09]];
	LOCAL CONST Robtarget Tr_meulage_bavure_P279 :=[[168.22253125,-27.6390078125,18.5],[0.259267363567836,-0.256875083353234,-0.655271217641931,0.661373765030723],[0,0,0,0],[8.999999E+09,8.999999E+09,8.999999E+09,8.999999E+09,8.999999E+09,8.999999E+09]];
	LOCAL CONST Robtarget Tr_meulage_bavure_P280 :=[[169.40265625,-28.78241015625,18.5],[0.258789906531584,-0.255569069163327,-0.654540181424425,0.662789096217828],[0,0,0,0],[8.999999E+09,8.999999E+09,8.999999E+09,8.999999E+09,8.999999E+09,8.999999E+09]];
	LOCAL CONST Robtarget Tr_meulage_bavure_P281 :=[[169.858453125,-29.2157890625,18.5],[0.258023081948368,-0.254048344297428,-0.653986108235206,0.6642181103952],[0,0,0,0],[8.999999E+09,8.999999E+09,8.999999E+09,8.999999E+09,8.999999E+09,8.999999E+09]];
	LOCAL CONST Robtarget Tr_meulage_bavure_P282 :=[[172.95453125,-32.14404296875,18.5],[0.256933979463729,-0.252301102255948,-0.653641483281607,0.665643970400683],[0,0,0,0],[8.999999E+09,8.999999E+09,8.999999E+09,8.999999E+09,8.999999E+09,8.999999E+09]];
	LOCAL CONST Robtarget Tr_meulage_bavure_P283 :=[[172.9580625,-32.147765625,18.5],[0.255677021101386,-0.250494831395092,-0.653464159645222,0.666982902617623],[0,0,0,0],[8.999999E+09,8.999999E+09,8.999999E+09,8.999999E+09,8.999999E+09,8.999999E+09]];
	LOCAL CONST Robtarget Tr_meulage_bavure_P284 :=[[172.978578125,-32.166748046875,18.5],[0.254606008805718,-0.24898304048042,-0.653332266113461,0.668086952340934],[0,0,0,0],[8.999999E+09,8.999999E+09,8.999999E+09,8.999999E+09,8.999999E+09,8.999999E+09]];
	LOCAL CONST Robtarget Tr_meulage_bavure_P285 :=[[176.13025,-35.13946484375,18.5],[0.25419766294075,-0.248233936654389,-0.653078752575925,0.668768722192059],[0,0,0,0],[8.999999E+09,8.999999E+09,8.999999E+09,8.999999E+09,8.999999E+09,8.999999E+09]];
	LOCAL CONST Robtarget Tr_meulage_bavure_P286 :=[[178.41265625,-37.24740625,18.5],[0.254822213405293,-0.248615062713904,-0.652581706230746,0.668874657047161],[0,0,0,0],[8.999999E+09,8.999999E+09,8.999999E+09,8.999999E+09,8.999999E+09,8.999999E+09]];
	LOCAL CONST Robtarget Tr_meulage_bavure_P287 :=[[179.163265625,-37.9834296875,18.5],[0.256531308956207,-0.250181631981869,-0.651828202631412,0.66837177738023],[0,0,0,0],[8.999999E+09,8.999999E+09,8.999999E+09,8.999999E+09,8.999999E+09,8.999999E+09]];
	LOCAL CONST Robtarget Tr_meulage_bavure_P288 :=[[183.01325,-41.69647265625,18.5],[0.258970472158777,-0.252580796254737,-0.650933258356023,0.667400276505183],[0,0,0,0],[8.999999E+09,8.999999E+09,8.999999E+09,8.999999E+09,8.999999E+09,8.999999E+09]];
	LOCAL CONST Robtarget Tr_meulage_bavure_P289 :=[[184.337828125,-43.04312109375,18.5],[0.261489652462882,-0.255175884048927,-0.650128348220494,0.666214350411925],[0,0,0,0],[8.999999E+09,8.999999E+09,8.999999E+09,8.999999E+09,8.999999E+09,8.999999E+09]];
	LOCAL CONST Robtarget Tr_meulage_bavure_P290 :=[[186.83959375,-45.2666640625,18.5],[0.263425364638095,-0.25732195683586,-0.649666485062982,0.665075894903252],[0,0,0,0],[8.999999E+09,8.999999E+09,8.999999E+09,8.999999E+09,8.999999E+09,8.999999E+09]];
	LOCAL CONST Robtarget Tr_meulage_bavure_P291 :=[[189.89825,-48.1846015625,18.5],[0.264397871423589,-0.258627663642258,-0.649677389784353,0.66417225656347],[0,0,0,0],[8.999999E+09,8.999999E+09,8.999999E+09,8.999999E+09,8.999999E+09,8.999999E+09]];
	LOCAL CONST Robtarget Tr_meulage_bavure_P292 :=[[191.546625,-49.80027734375,18.5],[0.264422475899701,-0.259089803919544,-0.650143979706336,0.663525457986061],[0,0,0,0],[8.999999E+09,8.999999E+09,8.999999E+09,8.999999E+09,8.999999E+09,8.999999E+09]];
	LOCAL CONST Robtarget Tr_meulage_bavure_P293 :=[[193.675234375,-51.7829140625,18.5],[0.263852745825249,-0.259032885988697,-0.650910852741964,0.663022438745155],[0,0,0,0],[8.999999E+09,8.999999E+09,8.999999E+09,8.999999E+09,8.999999E+09,8.999999E+09]];
	LOCAL CONST Robtarget Tr_meulage_bavure_P294 :=[[194.3465,-52.400453125,18.5],[0.263168525877941,-0.258905289316549,-0.651768847479954,0.662501130267563],[0,0,0,0],[8.999999E+09,8.999999E+09,8.999999E+09,8.999999E+09,8.999999E+09,8.999999E+09]];
	LOCAL CONST Robtarget Tr_meulage_bavure_P295 :=[[194.646234375,-52.6956484375,18.5],[0.262768608813241,-0.259081532332096,-0.652542503602902,0.661829055586459],[0,0,0,0],[8.999999E+09,8.999999E+09,8.999999E+09,8.999999E+09,8.999999E+09,8.999999E+09]];
	LOCAL CONST Robtarget Tr_meulage_bavure_P296 :=[[196.206296875,-54.1644453125,18.5],[0.262866437444509,-0.259752724255118,-0.653123903091844,0.660953043352819],[0,0,0,0],[8.999999E+09,8.999999E+09,8.999999E+09,8.999999E+09,8.999999E+09,8.999999E+09]];
	LOCAL CONST Robtarget Tr_meulage_bavure_P297 :=[[197.312078125,-55.3264140625,18.5],[0.263466001916206,-0.260914274673817,-0.653496503047982,0.659887662871329],[0,0,0,0],[8.999999E+09,8.999999E+09,8.999999E+09,8.999999E+09,8.999999E+09,8.999999E+09]];
	LOCAL CONST Robtarget Tr_meulage_bavure_P298 :=[[200.643,-58.4599296875,18.5],[0.264441619430254,-0.262431960028953,-0.653693514880082,0.658699388850628],[0,0,0,0],[8.999999E+09,8.999999E+09,8.999999E+09,8.999999E+09,8.999999E+09,8.999999E+09]];
	LOCAL CONST Robtarget Tr_meulage_bavure_P299 :=[[202.429203125,-60.06010546875,18.5],[0.265594055182714,-0.264098750804325,-0.653780473157078,0.657482121881427],[0,0,0,0],[8.999999E+09,8.999999E+09,8.999999E+09,8.999999E+09,8.999999E+09,8.999999E+09]];
	LOCAL CONST Robtarget Tr_meulage_bavure_P300 :=[[204.01825,-61.5348203125,18.5],[0.266724842073626,-0.265722189592481,-0.653841434802063,0.656308581929992],[0,0,0,0],[8.999999E+09,8.999999E+09,8.999999E+09,8.999999E+09,8.999999E+09,8.999999E+09]];
	LOCAL CONST Robtarget Tr_meulage_bavure_P301 :=[[206.714046875,-64.1923359375,18.5],[0.267671193043609,-0.267130213512057,-0.65393416937691,0.655258486068624],[0,0,0,0],[8.999999E+09,8.999999E+09,8.999999E+09,8.999999E+09,8.999999E+09,8.999999E+09]];
	LOCAL CONST Robtarget Tr_meulage_bavure_P302 :=[[207.529421875,-65.00823828125,18.5],[0.268272548438992,-0.26816981364774,-0.654135643214202,0.654386239982876],[0,0,0,0],[8.999999E+09,8.999999E+09,8.999999E+09,8.999999E+09,8.999999E+09,8.999999E+09]];
	LOCAL CONST Robtarget Tr_meulage_bavure_P303 :=[[208.419,-65.7788515625,18.5],[0.268392856729529,-0.268713815060226,-0.65451543484137,0.653733665651964],[0,0,0,0],[8.999999E+09,8.999999E+09,8.999999E+09,8.999999E+09,8.999999E+09,8.999999E+09]];
	LOCAL CONST Robtarget Tr_meulage_bavure_P304 :=[[209.78809375,-67.094375,18.5],[0.267897632221563,-0.268629907144974,-0.655135720065629,0.653349844976986],[0,0,0,0],[8.999999E+09,8.999999E+09,8.999999E+09,8.999999E+09,8.999999E+09,8.999999E+09]];
	LOCAL CONST Robtarget Tr_meulage_bavure_P305 :=[[212.06896875,-69.2288515625,18.5],[0.266662132875515,-0.267808956856003,-0.656067123294074,0.653257682121396],[0,0,0,0],[8.999999E+09,8.999999E+09,8.999999E+09,8.999999E+09,8.999999E+09,8.999999E+09]];
	LOCAL CONST Robtarget Tr_meulage_bavure_P306 :=[[213.341859375,-70.4299140625,18.5],[0.264634999925103,-0.266203868899579,-0.65733623565366,0.653462233257756],[0,0,0,0],[8.999999E+09,8.999999E+09,8.999999E+09,8.999999E+09,8.999999E+09,8.999999E+09]];
	LOCAL CONST Robtarget Tr_meulage_bavure_P307 :=[[214.866390625,-71.9375,18.5],[0.261877252030233,-0.263887216303028,-0.658928234244354,0.65390933932507],[0,0,0,0],[8.999999E+09,8.999999E+09,8.999999E+09,8.999999E+09,8.999999E+09,8.999999E+09]];
	LOCAL CONST Robtarget Tr_meulage_bavure_P308 :=[[216.273015625,-73.3049140625,18.5],[0.258610074877241,-0.261086458885015,-0.660756241414296,0.654489021749734],[0,0,0,0],[8.999999E+09,8.999999E+09,8.999999E+09,8.999999E+09,8.999999E+09,8.999999E+09]];
	LOCAL CONST Robtarget Tr_meulage_bavure_P309 :=[[217.93084375,-74.80875,18.5],[0.255187017422962,-0.258162739827659,-0.662682790903147,0.655044353112265],[0,0,0,0],[8.999999E+09,8.999999E+09,8.999999E+09,8.999999E+09,8.999999E+09,8.999999E+09]];
	LOCAL CONST Robtarget Tr_meulage_bavure_P310 :=[[219.9919375,-76.78784375,18.5],[0.252031870609241,-0.255546583538498,-0.664545020226845,0.655405062484804],[0,0,0,0],[8.999999E+09,8.999999E+09,8.999999E+09,8.999999E+09,8.999999E+09,8.999999E+09]];
	LOCAL CONST Robtarget Tr_meulage_bavure_P311 :=[[223.11303125,-79.7946640625,18.5],[0.249517437957387,-0.253625111272672,-0.66621152323485,0.655421663813615],[0,0,0,0],[8.999999E+09,8.999999E+09,8.999999E+09,8.999999E+09,8.999999E+09,8.999999E+09]];
	LOCAL CONST Robtarget Tr_meulage_bavure_P312 :=[[223.586671875,-80.2845,18.5],[0.247886123391458,-0.25264645461981,-0.667592271579042,0.655013585909429],[0,0,0,0],[8.999999E+09,8.999999E+09,8.999999E+09,8.999999E+09,8.999999E+09,8.999999E+09]];
	LOCAL CONST Robtarget Tr_meulage_bavure_P313 :=[[225.145453125,-81.6280078125,18.5],[0.247226187947275,-0.252706474255735,-0.668655494027861,0.654154783035829],[0,0,0,0],[8.999999E+09,8.999999E+09,8.999999E+09,8.999999E+09,8.999999E+09,8.999999E+09]];
	LOCAL CONST Robtarget Tr_meulage_bavure_P314 :=[[225.14734375,-81.6298046875,18.5],[0.247510922608473,-0.253773899671342,-0.669395777758071,0.652875519340992],[0,0,0,0],[8.999999E+09,8.999999E+09,8.999999E+09,8.999999E+09,8.999999E+09,8.999999E+09]];
	LOCAL CONST Robtarget Tr_meulage_bavure_P315 :=[[225.149046875,-81.631546875,18.5],[0.248619233556661,-0.255743201394327,-0.669863640626979,0.651203957767648],[0,0,0,0],[8.999999E+09,8.999999E+09,8.999999E+09,8.999999E+09,8.999999E+09,8.999999E+09]];
	LOCAL CONST Robtarget Tr_meulage_bavure_P316 :=[[225.157046875,-81.638796875,18.5],[0.250375365464276,-0.258437563266249,-0.670112796936134,0.649208011075084],[0,0,0,0],[8.999999E+09,8.999999E+09,8.999999E+09,8.999999E+09,8.999999E+09,8.999999E+09]];
	LOCAL CONST Robtarget Tr_meulage_bavure_P317 :=[[226.926515625,-83.3583203125,18.5],[0.252531351627815,-0.261605076541982,-0.670228144488434,0.646981402134623],[0,0,0,0],[8.999999E+09,8.999999E+09,8.999999E+09,8.999999E+09,8.999999E+09,8.999999E+09]];
	LOCAL CONST Robtarget Tr_meulage_bavure_P318 :=[[228.371453125,-84.7178203125,18.5],[0.254784045298984,-0.264935534336511,-0.670324056701176,0.644639365781047],[0,0,0,0],[8.999999E+09,8.999999E+09,8.999999E+09,8.999999E+09,8.999999E+09,8.999999E+09]];
	LOCAL CONST Robtarget Tr_meulage_bavure_P319 :=[[230.075921875,-86.4066953125,18.5],[0.256804586582402,-0.268105989181694,-0.670551527743567,0.642285942175224],[0,0,0,0],[8.999999E+09,8.999999E+09,8.999999E+09,8.999999E+09,8.999999E+09,8.999999E+09]];
	LOCAL CONST Robtarget Tr_meulage_bavure_P320 :=[[230.612359375,-86.89725,18.5],[0.258316794059642,-0.270836550896284,-0.67103971865786,0.640020072020349],[0,0,0,0],[8.999999E+09,8.999999E+09,8.999999E+09,8.999999E+09,8.999999E+09,8.999999E+09]];
	LOCAL CONST Robtarget Tr_meulage_bavure_P321 :=[[232.921875,-89.000765625,18.5],[0.259177064415251,-0.272976297599482,-0.671861183115027,0.637897907860849],[0,0,0,0],[8.999999E+09,8.999999E+09,8.999999E+09,8.999999E+09,8.999999E+09,8.999999E+09]];
	LOCAL CONST Robtarget Tr_meulage_bavure_P322 :=[[233.14696875,-89.230515625,18.5],[0.259346872555302,-0.274509337700894,-0.67307021074041,0.635893320160434],[0,0,0,0],[8.999999E+09,8.999999E+09,8.999999E+09,8.999999E+09,8.999999E+09,8.999999E+09]];
	LOCAL CONST Robtarget Tr_meulage_bavure_P323 :=[[233.633671875,-89.698046875,18.5],[0.258901562803361,-0.275527969766868,-0.674659043737541,0.63394754779656],[0,0,0,0],[8.999999E+09,8.999999E+09,8.999999E+09,8.999999E+09,8.999999E+09,8.999999E+09]];
	LOCAL CONST Robtarget Tr_meulage_bavure_P324 :=[[235.92975,-92.0232578125,18.5],[0.257979941652242,-0.276195294611128,-0.676591835090437,0.631969934117702],[0,0,0,0],[8.999999E+09,8.999999E+09,8.999999E+09,8.999999E+09,8.999999E+09,8.999999E+09]];
	LOCAL CONST Robtarget Tr_meulage_bavure_P325 :=[[237.01415625,-93.09296875,18.5],[0.256783789073463,-0.276749721697176,-0.678807289622409,0.629835169520638],[0,0,0,0],[8.999999E+09,8.999999E+09,8.999999E+09,8.999999E+09,8.999999E+09,8.999999E+09]];
	LOCAL CONST Robtarget Tr_meulage_bavure_P326 :=[[239.353453125,-95.390515625,18.5],[0.255565046936129,-0.277490809193132,-0.681220656298047,0.627394433375634],[0,0,0,0],[8.999999E+09,8.999999E+09,8.999999E+09,8.999999E+09,8.999999E+09,8.999999E+09]];
	LOCAL CONST Robtarget Tr_meulage_bavure_P327 :=[[240.431765625,-96.4383984375,18.5],[0.254634079752108,-0.278793589235626,-0.683719598449312,0.624470280098441],[0,0,0,0],[8.999999E+09,8.999999E+09,8.999999E+09,8.999999E+09,8.999999E+09,8.999999E+09]];
	LOCAL CONST Robtarget Tr_meulage_bavure_P328 :=[[242.6560625,-98.701796875,18.5],[0.254500785811857,-0.281251732062215,-0.686079311596363,0.620823639556849],[0,0,0,0],[8.999999E+09,8.999999E+09,8.999999E+09,8.999999E+09,8.999999E+09,8.999999E+09]];
	LOCAL CONST Robtarget Tr_meulage_bavure_P329 :=[[246.8254375,-102.681671875,18.5],[0.255842169953114,-0.285669943453742,-0.687974156953527,0.616140427861134],[0,0,0,0],[8.999999E+09,8.999999E+09,8.999999E+09,8.999999E+09,8.999999E+09,8.999999E+09]];
	LOCAL CONST Robtarget Tr_meulage_bavure_P330 :=[[248.599859375,-104.35665625,18.5],[0.259650589812881,-0.293261648786271,-0.688885285218938,0.609931340701397],[0,0,0,0],[8.999999E+09,8.999999E+09,8.999999E+09,8.999999E+09,8.999999E+09,8.999999E+09]];
	LOCAL CONST Robtarget Tr_meulage_bavure_P331 :=[[250.438234375,-106.0511171875,18.5],[0.267312128338324,-0.305740191459316,-0.687954426212445,0.60148638290851],[0,0,0,0],[8.999999E+09,8.999999E+09,8.999999E+09,8.999999E+09,8.999999E+09,8.999999E+09]];
	LOCAL CONST Robtarget Tr_meulage_bavure_P332 :=[[251.455265625,-106.9372109375,18.5],[0.280426723316242,-0.325176214800632,-0.683923695580389,0.58980476498729],[0,0,0,0],[8.999999E+09,8.999999E+09,8.999999E+09,8.999999E+09,8.999999E+09,8.999999E+09]];
	LOCAL CONST Robtarget Tr_meulage_bavure_P333 :=[[251.737359375,-107.2268359375,18.5],[0.300374422900762,-0.353505629810181,-0.675097094659343,0.573631317609191],[0,0,0,0],[8.999999E+09,8.999999E+09,8.999999E+09,8.999999E+09,8.999999E+09,8.999999E+09]];
	LOCAL CONST Robtarget Tr_meulage_bavure_P334 :=[[253.481390625,-108.6631015625,18.5],[0.32734997603317,-0.391411246462876,-0.659713687334042,0.55174004755644],[0,0,0,0],[8.999999E+09,8.999999E+09,8.999999E+09,8.999999E+09,8.999999E+09,8.999999E+09]];
	LOCAL CONST Robtarget Tr_meulage_bavure_P335 :=[[254.392390625,-109.8107109375,18.5],[0.359381630447848,-0.436998810608551,-0.636849590709484,0.523736080518156],[0,0,0,0],[8.999999E+09,8.999999E+09,8.999999E+09,8.999999E+09,8.999999E+09,8.999999E+09]];
	LOCAL CONST Robtarget Tr_meulage_bavure_P336 :=[[254.939140625,-110.3713046875,18.5],[0.392191537565192,-0.485371371703557,-0.607791994686316,0.491110293710169],[0,0,0,0],[8.999999E+09,8.999999E+09,8.999999E+09,8.999999E+09,8.999999E+09,8.999999E+09]];
	LOCAL CONST Robtarget Tr_meulage_bavure_P337 :=[[255.94690625,-112.398984375,18.5],[0.421112549399302,-0.53076465837811,-0.576173490924067,0.457140248186006],[0,0,0,0],[8.999999E+09,8.999999E+09,8.999999E+09,8.999999E+09,8.999999E+09,8.999999E+09]];
	LOCAL CONST Robtarget Tr_meulage_bavure_P338 :=[[256.09521875,-112.7145390625,18.5],[0.443682291515977,-0.569779282555571,-0.545780951921822,0.424994995129237],[0,0,0,0],[8.999999E+09,8.999999E+09,8.999999E+09,8.999999E+09,8.999999E+09,8.999999E+09]];
	LOCAL CONST Robtarget Tr_meulage_bavure_P339 :=[[256.072875,-112.91875,18.5],[0.460242390460929,-0.602382444020647,-0.51821544894664,0.395935703911069],[0,0,0,0],[8.999999E+09,8.999999E+09,8.999999E+09,8.999999E+09,8.999999E+09,8.999999E+09]];
	LOCAL CONST Robtarget Tr_meulage_bavure_P340 :=[[255.463875,-115.97734375,18.5],[0.472619163756135,-0.630494047982215,-0.492668488714996,0.369304944100041],[0,0,0,0],[8.999999E+09,8.999999E+09,8.999999E+09,8.999999E+09,8.999999E+09,8.999999E+09]];
	LOCAL CONST Robtarget Tr_meulage_bavure_P341 :=[[255.24884375,-116.269609375,18.5],[0.482648071257794,-0.656177098846216,-0.467278796586354,0.343704786876329],[0,0,0,0],[8.999999E+09,8.999999E+09,8.999999E+09,8.999999E+09,8.999999E+09,8.999999E+09]];
	LOCAL CONST Robtarget Tr_meulage_bavure_P342 :=[[253.679625,-118.490859375,18.5],[0.491311940362503,-0.680489101310208,-0.440766528698278,0.318232662425666],[0,0,0,0],[8.999999E+09,8.999999E+09,8.999999E+09,8.999999E+09,8.999999E+09,8.999999E+09]];
	LOCAL CONST Robtarget Tr_meulage_bavure_P343 :=[[251.1953125,-120.82340625,18.5],[0.49864002434769,-0.703211752973509,-0.413417834571171,0.293150218585871],[0,0,0,0],[8.999999E+09,8.999999E+09,8.999999E+09,8.999999E+09,8.999999E+09,8.999999E+09]];
	LOCAL CONST Robtarget Tr_meulage_bavure_P344 :=[[251.117125,-120.9000859375,18.5],[0.504155220019859,-0.723408002325757,-0.386997920580896,0.269705368437203],[0,0,0,0],[8.999999E+09,8.999999E+09,8.999999E+09,8.999999E+09,8.999999E+09,8.999999E+09]];
	LOCAL CONST Robtarget Tr_meulage_bavure_P345 :=[[251.042171875,-120.9748828125,18.5],[0.507539751954385,-0.740341339980761,-0.36356250267342,0.249239658063101],[0,0,0,0],[8.999999E+09,8.999999E+09,8.999999E+09,8.999999E+09,8.999999E+09,8.999999E+09]];
	LOCAL CONST Robtarget Tr_meulage_bavure_P346 :=[[245.482234375,-126.893171875,18.5],[0.508977984051693,-0.753994398290478,-0.344173981965959,0.232331937612871],[0,0,0,0],[8.999999E+09,8.999999E+09,8.999999E+09,8.999999E+09,8.999999E+09,8.999999E+09]];
	LOCAL CONST Robtarget Tr_meulage_bavure_P347 :=[[244.61303125,-127.7652265625,18.5],[0.509015155882975,-0.764923836834545,-0.328602716427865,0.218667212174064],[0,0,0,0],[8.999999E+09,8.999999E+09,8.999999E+09,8.999999E+09,8.999999E+09,8.999999E+09]];
	LOCAL CONST Robtarget Tr_meulage_bavure_P348 :=[[239.66028125,-132.926609375,18.5],[0.508291212967999,-0.77392261521099,-0.31572895091285,0.207362142253531],[0,0,0,0],[8.999999E+09,8.999999E+09,8.999999E+09,8.999999E+09,8.999999E+09,8.999999E+09]];
	LOCAL CONST Robtarget Tr_meulage_bavure_P349 :=[[239.622796875,-132.9660625,18.5],[0.507282243450708,-0.781611571950647,-0.304467011469221,0.197605452858611],[0,0,0,0],[8.999999E+09,8.999999E+09,8.999999E+09,8.999999E+09,8.999999E+09,8.999999E+09]];
	LOCAL CONST Robtarget Tr_meulage_bavure_P350 :=[[236.968390625,-135.39278125,18.5],[0.50620477642001,-0.788265747252369,-0.29437613318859,0.189041075555462],[0,0,0,0],[8.999999E+09,8.999999E+09,8.999999E+09,8.999999E+09,8.999999E+09,8.999999E+09]];
	LOCAL CONST Robtarget Tr_meulage_bavure_P351 :=[[236.60265625,-135.67,18.5],[0.505042321602662,-0.793832060283945,-0.285824608359756,0.181843907545821],[0,0,0,0],[8.999999E+09,8.999999E+09,8.999999E+09,8.999999E+09,8.999999E+09,8.999999E+09]];
	LOCAL CONST Robtarget Tr_meulage_bavure_P352 :=[[234.39875,-137.287734375,18.5],[0.503664362651905,-0.798097785279606,-0.279665579612292,0.176491638630162],[0,0,0,0],[8.999999E+09,8.999999E+09,8.999999E+09,8.999999E+09,8.999999E+09,8.999999E+09]];
	LOCAL CONST Robtarget Tr_meulage_bavure_P353 :=[[230.26465625,-139.943578125,18.5],[0.50195967306889,-0.800878747388832,-0.276687889066687,0.173417215515903],[0,0,0,0],[8.999999E+09,8.999999E+09,8.999999E+09,8.999999E+09,8.999999E+09,8.999999E+09]];
	LOCAL CONST Robtarget Tr_meulage_bavure_P354 :=[[230.14325,-140.029359375,18.5],[0.499867033670729,-0.80210964869429,-0.277292509785057,0.172806030386248],[0,0,0,0],[8.999999E+09,8.999999E+09,8.999999E+09,8.999999E+09,8.999999E+09,8.999999E+09]];
	LOCAL CONST Robtarget Tr_meulage_bavure_P355 :=[[230.00421875,-140.136453125,18.5],[0.497437845999554,-0.801925647704508,-0.281163711390674,0.174407030586647],[0,0,0,0],[8.999999E+09,8.999999E+09,8.999999E+09,8.999999E+09,8.999999E+09,8.999999E+09]];
	LOCAL CONST Robtarget Tr_meulage_bavure_P356 :=[[229.714359375,-140.400703125,18.5],[0.494837978091229,-0.800644221482799,-0.287341980224137,0.177591645202296],[0,0,0,0],[8.999999E+09,8.999999E+09,8.999999E+09,8.999999E+09,8.999999E+09,8.999999E+09]];
	LOCAL CONST Robtarget Tr_meulage_bavure_P357 :=[[226.640875,-143.141875,18.5],[0.49230591751571,-0.798722201939685,-0.294497477439139,0.181518493519585],[0,0,0,0],[8.999999E+09,8.999999E+09,8.999999E+09,8.999999E+09,8.999999E+09,8.999999E+09]];
	LOCAL CONST Robtarget Tr_meulage_bavure_P358 :=[[223.423890625,-146.300015625,18.5],[0.490095172220216,-0.796653988112918,-0.30131216676978,0.185364839024883],[0,0,0,0],[8.999999E+09,8.999999E+09,8.999999E+09,8.999999E+09,8.999999E+09,8.999999E+09]];
	LOCAL CONST Robtarget Tr_meulage_bavure_P359 :=[[221.904171875,-147.811015625,18.5],[0.48839504006106,-0.794840743506669,-0.30684050435915,0.188540134162845],[0,0,0,0],[8.999999E+09,8.999999E+09,8.999999E+09,8.999999E+09,8.999999E+09,8.999999E+09]];
	LOCAL CONST Robtarget Tr_meulage_bavure_P360 :=[[218.185359375,-151.3090625,18.5],[0.487282774655116,-0.793495177884697,-0.310678764764617,0.190786805944427],[0,0,0,0],[8.999999E+09,8.999999E+09,8.999999E+09,8.999999E+09,8.999999E+09,8.999999E+09]];
	LOCAL CONST Robtarget Tr_meulage_bavure_P361 :=[[216.812140625,-152.594234375,18.5],[0.486723759757224,-0.79262793412152,-0.312919248812848,0.192152240321176],[0,0,0,0],[8.999999E+09,8.999999E+09,8.999999E+09,8.999999E+09,8.999999E+09,8.999999E+09]];
	LOCAL CONST Robtarget Tr_meulage_bavure_P362 :=[[212.958734375,-156.199421875,18.5],[0.4865930563528,-0.792124507031133,-0.313959203447844,0.192861560297329],[0,0,0,0],[8.999999E+09,8.999999E+09,8.999999E+09,8.999999E+09,8.999999E+09,8.999999E+09]];
	LOCAL CONST Robtarget Tr_meulage_bavure_P363 :=[[212.00659375,-157.107359375,18.5],[0.486746054524811,-0.791814814192313,-0.314293170704144,0.193202953597657],[0,0,0,0],[8.999999E+09,8.999999E+09,8.999999E+09,8.999999E+09,8.999999E+09,8.999999E+09]];
	LOCAL CONST Robtarget Tr_meulage_bavure_P364 :=[[207.901484375,-161.032171875,18.5],[0.487054530536913,-0.791544611083213,-0.314356154393915,0.193430145383962],[0,0,0,0],[8.999999E+09,8.999999E+09,8.999999E+09,8.999999E+09,8.999999E+09,8.999999E+09]];
	LOCAL CONST Robtarget Tr_meulage_bavure_P365 :=[[206.57665625,-162.19796875,18.5],[0.487428648832311,-0.791227006975657,-0.314414411664529,0.19369231649061],[0,0,0,0],[8.999999E+09,8.999999E+09,8.999999E+09,8.999999E+09,8.999999E+09,8.999999E+09]];
	LOCAL CONST Robtarget Tr_meulage_bavure_P366 :=[[205.275140625,-163.26084375,18.5],[0.487832381924595,-0.790849886594734,-0.314535187261225,0.194019689705502],[0,0,0,0],[8.999999E+09,8.999999E+09,8.999999E+09,8.999999E+09,8.999999E+09,8.999999E+09]];
	LOCAL CONST Robtarget Tr_meulage_bavure_P367 :=[[201.602234375,-166.729296875,18.5],[0.488271998186391,-0.79046796223385,-0.314616301991688,0.194338465029464],[0,0,0,0],[8.999999E+09,8.999999E+09,8.999999E+09,8.999999E+09,8.999999E+09,8.999999E+09]];
	LOCAL CONST Robtarget Tr_meulage_bavure_P368 :=[[199.991703125,-168.0753125,18.5],[0.488795182935565,-0.790183552553002,-0.314420997271817,0.194495909695554],[0,0,0,0],[8.999999E+09,8.999999E+09,8.999999E+09,8.999999E+09,8.999999E+09,8.999999E+09]];
	LOCAL CONST Robtarget Tr_meulage_bavure_P369 :=[[198.935546875,-169.07909375,18.5],[0.489454789053762,-0.790096187963527,-0.313710271490623,0.194339622308783],[0,0,0,0],[8.999999E+09,8.999999E+09,8.999999E+09,8.999999E+09,8.999999E+09,8.999999E+09]];
	LOCAL CONST Robtarget Tr_meulage_bavure_P370 :=[[197.601015625,-170.208640625,18.5],[0.4902673605879,-0.790261060519044,-0.312365063823061,0.193787095216128],[0,0,0,0],[8.999999E+09,8.999999E+09,8.999999E+09,8.999999E+09,8.999999E+09,8.999999E+09]];
	LOCAL CONST Robtarget Tr_meulage_bavure_P371 :=[[193.895015625,-173.436875,18.5],[0.491219421636612,-0.790658854998606,-0.310428762271124,0.192862744909699],[0,0,0,0],[8.999999E+09,8.999999E+09,8.999999E+09,8.999999E+09,8.999999E+09,8.999999E+09]];
	LOCAL CONST Robtarget Tr_meulage_bavure_P372 :=[[192.234921875,-174.862109375,18.5],[0.492256801861418,-0.791205515278538,-0.308108553537469,0.191692965053597],[0,0,0,0],[8.999999E+09,8.999999E+09,8.999999E+09,8.999999E+09,8.999999E+09,8.999999E+09]];
	LOCAL CONST Robtarget Tr_meulage_bavure_P373 :=[[188.893734375,-177.886859375,18.5],[0.493301322129992,-0.791771061133922,-0.305728476679111,0.190479633775204],[0,0,0,0],[8.999999E+09,8.999999E+09,8.999999E+09,8.999999E+09,8.999999E+09,8.999999E+09]];
	LOCAL CONST Robtarget Tr_meulage_bavure_P374 :=[[188.0365,-178.692109375,18.5],[0.494273725890403,-0.792210607412543,-0.303650350104771,0.189452638616404],[0,0,0,0],[8.999999E+09,8.999999E+09,8.999999E+09,8.999999E+09,8.999999E+09,8.999999E+09]];
	LOCAL CONST Robtarget Tr_meulage_bavure_P375 :=[[187.765984375,-178.90815625,18.5],[0.495097371215471,-0.792404064595417,-0.302197782362455,0.188814437380742],[0,0,0,0],[8.999999E+09,8.999999E+09,8.999999E+09,8.999999E+09,8.999999E+09,8.999999E+09]];
	LOCAL CONST Robtarget Tr_meulage_bavure_P376 :=[[185.5340625,-180.671125,18.5],[0.495730291199621,-0.792283183296903,-0.301557792251133,0.188684217105424],[0,0,0,0],[8.999999E+09,8.999999E+09,8.999999E+09,8.999999E+09,8.999999E+09,8.999999E+09]];
	LOCAL CONST Robtarget Tr_meulage_bavure_P377 :=[[181.474421875,-183.969875,18.5],[0.496182391256916,-0.791854309210816,-0.301709363872902,0.189053556809279],[0,0,0,0],[8.999999E+09,8.999999E+09,8.999999E+09,8.999999E+09,8.999999E+09,8.999999E+09]];
	LOCAL CONST Robtarget Tr_meulage_bavure_P378 :=[[179.5496875,-185.64784375,18.5],[0.496509502715142,-0.791209538572831,-0.302410651330606,0.189772436741295],[0,0,0,0],[8.999999E+09,8.999999E+09,8.999999E+09,8.999999E+09,8.999999E+09,8.999999E+09]];
	LOCAL CONST Robtarget Tr_meulage_bavure_P379 :=[[176.253421875,-188.743984375,18.5],[0.496813240459927,-0.790495699371747,-0.3032606231187,0.190594196774555],[0,0,0,0],[8.999999E+09,8.999999E+09,8.999999E+09,8.999999E+09,8.999999E+09,8.999999E+09]];
	LOCAL CONST Robtarget Tr_meulage_bavure_P380 :=[[173.68871875,-191.181796875,18.5],[0.497179338438338,-0.789866020919361,-0.303873632232921,0.191272554384059],[0,0,0,0],[8.999999E+09,8.999999E+09,8.999999E+09,8.999999E+09,8.999999E+09,8.999999E+09]];
	LOCAL CONST Robtarget Tr_meulage_bavure_P381 :=[[171.9218125,-192.6625625,18.5],[0.497658682619734,-0.789408606721568,-0.304029537052258,0.191666188585502],[0,0,0,0],[8.999999E+09,8.999999E+09,8.999999E+09,8.999999E+09,8.999999E+09,8.999999E+09]];
	LOCAL CONST Robtarget Tr_meulage_bavure_P382 :=[[171.007453125,-193.46353125,18.5],[0.498245184649095,-0.789123410886627,-0.303738769813775,0.191777835206939],[0,0,0,0],[8.999999E+09,8.999999E+09,8.999999E+09,8.999999E+09,8.999999E+09,8.999999E+09]];
	LOCAL CONST Robtarget Tr_meulage_bavure_P383 :=[[166.679078125,-197.012984375,18.5],[0.498886589522245,-0.78894556785478,-0.303185226164459,0.191717970969778],[0,0,0,0],[8.999999E+09,8.999999E+09,8.999999E+09,8.999999E+09,8.999999E+09,8.999999E+09]];
	LOCAL CONST Robtarget Tr_meulage_bavure_P384 :=[[165.283265625,-198.272703125,18.5],[0.499527176416304,-0.788795720298483,-0.302582420865105,0.191618867139341],[0,0,0,0],[8.999999E+09,8.999999E+09,8.999999E+09,8.999999E+09,8.999999E+09,8.999999E+09]];
	LOCAL CONST Robtarget Tr_meulage_bavure_P385 :=[[163.275640625,-200.049078125,18.5],[0.500132433755617,-0.788638359858759,-0.302039183489981,0.191544819041592],[0,0,0,0],[8.999999E+09,8.999999E+09,8.999999E+09,8.999999E+09,8.999999E+09,8.999999E+09]];
	LOCAL CONST Robtarget Tr_meulage_bavure_P386 :=[[162.551875,-200.721390625,18.5],[0.500699054016695,-0.788500566350645,-0.301512798400373,0.19146108370182],[0,0,0,0],[8.999999E+09,8.999999E+09,8.999999E+09,8.999999E+09,8.999999E+09,8.999999E+09]];
	LOCAL CONST Robtarget Tr_meulage_bavure_P387 :=[[160.374515625,-202.7565,18.5],[0.501256484122499,-0.788440419657543,-0.300861444768358,0.19127475742315],[0,0,0,0],[8.999999E+09,8.999999E+09,8.999999E+09,8.999999E+09,8.999999E+09,8.999999E+09]];
	LOCAL CONST Robtarget Tr_meulage_bavure_P388 :=[[156.98296875,-205.7069375,18.5],[0.501825906227627,-0.788517881473655,-0.299950123784418,0.19089325204635],[0,0,0,0],[8.999999E+09,8.999999E+09,8.999999E+09,8.999999E+09,8.999999E+09,8.999999E+09]];
	LOCAL CONST Robtarget Tr_meulage_bavure_P389 :=[[155.02246875,-207.407171875,18.5],[0.5024198798864,-0.788752636326791,-0.298724645431767,0.190281710088324],[0,0,0,0],[8.999999E+09,8.999999E+09,8.999999E+09,8.999999E+09,8.999999E+09,8.999999E+09]];
	LOCAL CONST Robtarget Tr_meulage_bavure_P390 :=[[154.74103125,-207.667015625,18.5],[0.503013226773045,-0.789129609712322,-0.297242401248227,0.189470598423173],[0,0,0,0],[8.999999E+09,8.999999E+09,8.999999E+09,8.999999E+09,8.999999E+09,8.999999E+09]];
	LOCAL CONST Robtarget Tr_meulage_bavure_P391 :=[[154.18128125,-208.128484375,18.5],[0.503570788245277,-0.789602482706657,-0.295630527947991,0.188539044960733],[0,0,0,0],[8.999999E+09,8.999999E+09,8.999999E+09,8.999999E+09,8.999999E+09,8.999999E+09]];
	LOCAL CONST Robtarget Tr_meulage_bavure_P392 :=[[150.88921875,-210.8240625,18.5],[0.504063353783831,-0.790120332507248,-0.294018620041277,0.1875714439883],[0,0,0,0],[8.999999E+09,8.999999E+09,8.999999E+09,8.999999E+09,8.999999E+09,8.999999E+09]];
	LOCAL CONST Robtarget Tr_meulage_bavure_P393 :=[[147.99878125,-213.351421875,18.5],[0.504466664271247,-0.790651570405701,-0.292497321677643,0.186624745587087],[0,0,0,0],[8.999999E+09,8.999999E+09,8.999999E+09,8.999999E+09,8.999999E+09,8.999999E+09]];
	LOCAL CONST Robtarget Tr_meulage_bavure_P394 :=[[147.30334375,-213.979796875,18.5],[0.50478591123791,-0.791183787506578,-0.291083086543829,0.185714929207581],[0,0,0,0],[8.999999E+09,8.999999E+09,8.999999E+09,8.999999E+09,8.999999E+09,8.999999E+09]];
	LOCAL CONST Robtarget Tr_meulage_bavure_P395 :=[[146.075078125,-215.03696875,18.5],[0.505032444604601,-0.791732283743101,-0.289733199080166,0.184815838407881],[0,0,0,0],[8.999999E+09,8.999999E+09,8.999999E+09,8.999999E+09,8.999999E+09,8.999999E+09]];
	LOCAL CONST Robtarget Tr_meulage_bavure_P396 :=[[142.226375,-218.315546875,18.5],[0.505236705639819,-0.792314907457371,-0.288372314487386,0.183886831861958],[0,0,0,0],[8.999999E+09,8.999999E+09,8.999999E+09,8.999999E+09,8.999999E+09,8.999999E+09]];
	LOCAL CONST Robtarget Tr_meulage_bavure_P397 :=[[139.599859375,-220.624203125,18.5],[0.505417722762261,-0.792951043495939,-0.286936837101092,0.182890184676304],[0,0,0,0],[8.999999E+09,8.999999E+09,8.999999E+09,8.999999E+09,8.999999E+09,8.999999E+09]];
	LOCAL CONST Robtarget Tr_meulage_bavure_P398 :=[[135.929875,-223.670421875,18.5],[0.505583701554726,-0.793643228933096,-0.285408608866128,0.181817138565024],[0,0,0,0],[8.999999E+09,8.999999E+09,8.999999E+09,8.999999E+09,8.999999E+09,8.999999E+09]];
	LOCAL CONST Robtarget Tr_meulage_bavure_P399 :=[[135.325015625,-224.17259375,18.5],[0.505742041446702,-0.794367507520902,-0.283820133599593,0.18069693487124],[0,0,0,0],[8.999999E+09,8.999999E+09,8.999999E+09,8.999999E+09,8.999999E+09,8.999999E+09]];
	LOCAL CONST Robtarget Tr_meulage_bavure_P400 :=[[134.375484375,-225.0266875,18.5],[0.505882570871051,-0.795081685271838,-0.28226491384761,0.17959525785719],[0,0,0,0],[8.999999E+09,8.999999E+09,8.999999E+09,8.999999E+09,8.999999E+09,8.999999E+09]];
	LOCAL CONST Robtarget Tr_meulage_bavure_P401 :=[[132.353828125,-226.560765625,18.5],[0.505967586647417,-0.795719103642701,-0.28092568199914,0.178629982235803],[0,0,0,0],[8.999999E+09,8.999999E+09,8.999999E+09,8.999999E+09,8.999999E+09,8.999999E+09]];
	LOCAL CONST Robtarget Tr_meulage_bavure_P402 :=[[129.9619140625,-228.491734375,18.5],[0.505959204436771,-0.796178727061283,-0.280055484382664,0.17797090685833],[0,0,0,0],[8.999999E+09,8.999999E+09,8.999999E+09,8.999999E+09,8.999999E+09,8.999999E+09]];
	LOCAL CONST Robtarget Tr_meulage_bavure_P403 :=[[128.776609375,-229.421546875,18.5],[0.505777887213406,-0.796335227361326,-0.280016493263752,0.177847400795176],[0,0,0,0],[8.999999E+09,8.999999E+09,8.999999E+09,8.999999E+09,8.999999E+09,8.999999E+09]];
	LOCAL CONST Robtarget Tr_meulage_bavure_P404 :=[[125.57665625,-231.903484375,18.5],[0.505336309935758,-0.796022769150812,-0.281253936828837,0.178547438716621],[0,0,0,0],[8.999999E+09,8.999999E+09,8.999999E+09,8.999999E+09,8.999999E+09,8.999999E+09]];
	LOCAL CONST Robtarget Tr_meulage_bavure_P405 :=[[124.012875,-233.175625,18.5],[0.504547452682693,-0.795088661222945,-0.284163583525559,0.180324559015191],[0,0,0,0],[8.999999E+09,8.999999E+09,8.999999E+09,8.999999E+09,8.999999E+09,8.999999E+09]];
	LOCAL CONST Robtarget Tr_meulage_bavure_P406 :=[[119.8265390625,-236.527484375,18.5],[0.503370468355213,-0.793439914734652,-0.288919192011634,0.18329477292347],[0,0,0,0],[8.999999E+09,8.999999E+09,8.999999E+09,8.999999E+09,8.999999E+09,8.999999E+09]];
	LOCAL CONST Robtarget Tr_meulage_bavure_P407 :=[[115.14325,-240.122015625,18.5],[0.501858311895025,-0.791135780369372,-0.295239652306469,0.1872857696334],[0,0,0,0],[8.999999E+09,8.999999E+09,8.999999E+09,8.999999E+09,8.999999E+09,8.999999E+09]];
	LOCAL CONST Robtarget Tr_meulage_bavure_P408 :=[[112.6598515625,-242.025875,18.5],[0.500182721206282,-0.788448270007736,-0.302303954583065,0.191778231225359],[0,0,0,0],[8.999999E+09,8.999999E+09,8.999999E+09,8.999999E+09,8.999999E+09,8.999999E+09]];
	LOCAL CONST Robtarget Tr_meulage_bavure_P409 :=[[111.1560703125,-243.375359375,18.5],[0.49865267394023,-0.785828750124568,-0.308874382032093,0.195998220334296],[0,0,0,0],[8.999999E+09,8.999999E+09,8.999999E+09,8.999999E+09,8.999999E+09,8.999999E+09]];
	LOCAL CONST Robtarget Tr_meulage_bavure_P410 :=[[110.3673125,-244.039375,18.5],[0.497621591298346,-0.783792023832111,-0.313664158872072,0.1991421871175],[0,0,0,0],[8.999999E+09,8.999999E+09,8.999999E+09,8.999999E+09,8.999999E+09,8.999999E+09]];
	LOCAL CONST Robtarget Tr_meulage_bavure_P411 :=[[109.8060625,-244.531375,18.5],[0.497354907335162,-0.782726197952075,-0.31577999393736,0.200650917311739],[0,0,0,0],[8.999999E+09,8.999999E+09,8.999999E+09,8.999999E+09,8.999999E+09,8.999999E+09]];
	LOCAL CONST Robtarget Tr_meulage_bavure_P412 :=[[109.602328125,-244.825078125,18.5],[0.497955453435675,-0.782741193092734,-0.314970821619332,0.200374580618092],[0,0,0,0],[8.999999E+09,8.999999E+09,8.999999E+09,8.999999E+09,8.999999E+09,8.999999E+09]];
	LOCAL CONST Robtarget Tr_meulage_bavure_P413 :=[[108.86190625,-245.664390625,18.5],[0.499344601082734,-0.783654513474088,-0.311626607573442,0.19856845251319],[0,0,0,0],[8.999999E+09,8.999999E+09,8.999999E+09,8.999999E+09,8.999999E+09,8.999999E+09]];
	LOCAL CONST Robtarget Tr_meulage_bavure_P414 :=[[107.36975,-247.324296875,18.5],[0.501333101211148,-0.785100115983544,-0.306540508095392,0.195744339405403],[0,0,0,0],[8.999999E+09,8.999999E+09,8.999999E+09,8.999999E+09,8.999999E+09,8.999999E+09]];
	LOCAL CONST Robtarget Tr_meulage_bavure_P415 :=[[106.047390625,-248.54209375,18.5],[0.503713308995406,-0.786693032517252,-0.300577847762903,0.192457611862793],[0,0,0,0],[8.999999E+09,8.999999E+09,8.999999E+09,8.999999E+09,8.999999E+09,8.999999E+09]];
	LOCAL CONST Robtarget Tr_meulage_bavure_P416 :=[[104.331875,-249.96678125,18.5],[0.506344461347547,-0.788128255147287,-0.294427948180466,0.189159517950845],[0,0,0,0],[8.999999E+09,8.999999E+09,8.999999E+09,8.999999E+09,8.999999E+09,8.999999E+09]];
	LOCAL CONST Robtarget Tr_meulage_bavure_P417 :=[[103.2576015625,-250.858703125,18.5],[0.509174977923552,-0.789238842160337,-0.28846104843407,0.186099745884508],[0,0,0,0],[8.999999E+09,8.999999E+09,8.999999E+09,8.999999E+09,8.999999E+09,8.999999E+09]];
	LOCAL CONST Robtarget Tr_meulage_bavure_P418 :=[[102.75915625,-251.2904375,18.5],[0.512218586545232,-0.789981301336621,-0.282753779514576,0.183335657487371],[0,0,0,0],[8.999999E+09,8.999999E+09,8.999999E+09,8.999999E+09,8.999999E+09,8.999999E+09]];
	LOCAL CONST Robtarget Tr_meulage_bavure_P419 :=[[101.55465625,-252.2634375,18.5],[0.515558178968573,-0.790392695182263,-0.277131941008823,0.18076791411589],[0,0,0,0],[8.999999E+09,8.999999E+09,8.999999E+09,8.999999E+09,8.999999E+09,8.999999E+09]];
	LOCAL CONST Robtarget Tr_meulage_bavure_P420 :=[[96.767640625,-256.080875,18.5],[0.519319601635706,-0.790608076452266,-0.271151661356174,0.178108947976134],[0,0,0,0],[8.999999E+09,8.999999E+09,8.999999E+09,8.999999E+09,8.999999E+09,8.999999E+09]];
	LOCAL CONST Robtarget Tr_meulage_bavure_P421 :=[[95.7014765625,-256.787359375,18.5],[0.523646736830499,-0.790792621031918,-0.26424306451726,0.174976365211897],[0,0,0,0],[8.999999E+09,8.999999E+09,8.999999E+09,8.999999E+09,8.999999E+09,8.999999E+09]];
	LOCAL CONST Robtarget Tr_meulage_bavure_P422 :=[[92.0549296875,-259.538640625,18.5],[0.528699963003502,-0.791082270160416,-0.255806867411302,0.170962093878014],[0,0,0,0],[8.999999E+09,8.999999E+09,8.999999E+09,8.999999E+09,8.999999E+09,8.999999E+09]];
	LOCAL CONST Robtarget Tr_meulage_bavure_P423 :=[[91.4923125,-259.97546875,18.5],[0.534608568869989,-0.79162578546872,-0.245170462595784,0.165570945948809],[0,0,0,0],[8.999999E+09,8.999999E+09,8.999999E+09,8.999999E+09,8.999999E+09,8.999999E+09]];
	LOCAL CONST Robtarget Tr_meulage_bavure_P424 :=[[88.78128125,-262.2035625,18.5],[0.541484313954335,-0.792528271325416,-0.231623519528993,0.158253663756491],[0,0,0,0],[8.999999E+09,8.999999E+09,8.999999E+09,8.999999E+09,8.999999E+09,8.999999E+09]];
	LOCAL CONST Robtarget Tr_meulage_bavure_P425 :=[[87.167421875,-263.531,18.5],[0.549468958690359,-0.793945751724411,-0.214005182825569,0.148107354571905],[0,0,0,0],[8.999999E+09,8.999999E+09,8.999999E+09,8.999999E+09,8.999999E+09,8.999999E+09]];
	LOCAL CONST Robtarget Tr_meulage_bavure_P426 :=[[86.8817109375,-263.7433125,18.5],[0.558759879050772,-0.796108517988154,-0.190203164461304,0.133496746697357],[0,0,0,0],[8.999999E+09,8.999999E+09,8.999999E+09,8.999999E+09,8.999999E+09,8.999999E+09]];
	LOCAL CONST Robtarget Tr_meulage_bavure_P427 :=[[84.4164453125,-265.018625,18.5],[0.569472736870233,-0.799114473607361,-0.156894536364773,0.111807712129531],[0,0,0,0],[8.999999E+09,8.999999E+09,8.999999E+09,8.999999E+09,8.999999E+09,8.999999E+09]];
	LOCAL CONST Robtarget Tr_meulage_bavure_P428 :=[[83.8686796875,-265.19353125,18.5],[0.581212823884327,-0.802373504228919,-0.109819349384467,0.079549503861328],[0,0,0,0],[8.999999E+09,8.999999E+09,8.999999E+09,8.999999E+09,8.999999E+09,8.999999E+09]];
	LOCAL CONST Robtarget Tr_meulage_bavure_P429 :=[[82.6865546875,-265.43353125,18.5],[0.592369753025986,-0.803669610990369,-0.0456296839927781,0.0336327817648186],[0,0,0,0],[8.999999E+09,8.999999E+09,8.999999E+09,8.999999E+09,8.999999E+09,8.999999E+09]];
	LOCAL CONST Robtarget Tr_meulage_bavure_P430 :=[[81.7553125,-265.35940625,18.5],[0.599826724811674,-0.798998986380909,0.034009555252823,-0.0255317472078459],[0,0,0,0],[8.999999E+09,8.999999E+09,8.999999E+09,8.999999E+09,8.999999E+09,8.999999E+09]];
	LOCAL CONST Robtarget Tr_meulage_bavure_P431 :=[[80.5024375,-265.07528125,18.5],[0.600919493093,-0.785241592837045,0.118567943424758,-0.0907361366359396],[0,0,0,0],[8.999999E+09,8.999999E+09,8.999999E+09,8.999999E+09,8.999999E+09,8.999999E+09]];
	LOCAL CONST Robtarget Tr_meulage_bavure_P432 :=[[78.1274375,-263.5239375,18.5],[0.596620029296442,-0.764221720302449,0.193093844588129,-0.150746376548339],[0,0,0,0],[8.999999E+09,8.999999E+09,8.999999E+09,8.999999E+09,8.999999E+09,8.999999E+09]];
	LOCAL CONST Robtarget Tr_meulage_bavure_P433 :=[[77.7958359375,-263.26696875,18.5],[0.590897553034023,-0.741452793725075,0.24864190713248,-0.19815407771027],[0,0,0,0],[8.999999E+09,8.999999E+09,8.999999E+09,8.999999E+09,8.999999E+09,8.999999E+09]];
	LOCAL CONST Robtarget Tr_meulage_bavure_P434 :=[[77.0217578125,-262.36253125,18.5],[0.587093406891487,-0.721273172698127,0.285048737783321,-0.232020600418711],[0,0,0,0],[8.999999E+09,8.999999E+09,8.999999E+09,8.999999E+09,8.999999E+09,8.999999E+09]];
	LOCAL CONST Robtarget Tr_meulage_bavure_P435 :=[[75.792453125,-260.825625,18.5],[0.586466915212699,-0.705162675703012,0.306385665239911,-0.25481362265736],[0,0,0,0],[8.999999E+09,8.999999E+09,8.999999E+09,8.999999E+09,8.999999E+09,8.999999E+09]];
	LOCAL CONST Robtarget Tr_meulage_bavure_P436 :=[[74.9748515625,-259.83715625,18.5],[0.58882301322574,-0.692745445378461,0.317275986857442,-0.269679727022248],[0,0,0,0],[8.999999E+09,8.999999E+09,8.999999E+09,8.999999E+09,8.999999E+09,8.999999E+09]];
	LOCAL CONST Robtarget Tr_meulage_bavure_P437 :=[[73.37878125,-257.411125,18.5],[0.593361712396459,-0.682960125008683,0.321592434747235,-0.279402311771774],[0,0,0,0],[8.999999E+09,8.999999E+09,8.999999E+09,8.999999E+09,8.999999E+09,8.999999E+09]];
	LOCAL CONST Robtarget Tr_meulage_bavure_P438 :=[[71.870421875,-255.23596875,18.5],[0.599133760764523,-0.674688291952299,0.322336821815463,-0.28624014169322],[0,0,0,0],[8.999999E+09,8.999999E+09,8.999999E+09,8.999999E+09,8.999999E+09,8.999999E+09]];
	LOCAL CONST Robtarget Tr_meulage_bavure_P439 :=[[71.1931484375,-254.256984375,18.5],[0.605313110472779,-0.667005715123286,0.321679908392056,-0.291927132722399],[0,0,0,0],[8.999999E+09,8.999999E+09,8.999999E+09,8.999999E+09,8.999999E+09,8.999999E+09]];
	LOCAL CONST Robtarget Tr_meulage_bavure_P440 :=[[69.68765625,-252.447578125,18.5],[0.611257667347024,-0.659330126193572,0.321036635445154,-0.297629513834059],[0,0,0,0],[8.999999E+09,8.999999E+09,8.999999E+09,8.999999E+09,8.999999E+09,8.999999E+09]];
	LOCAL CONST Robtarget Tr_meulage_bavure_P441 :=[[69.1363515625,-251.749515625,18.5],[0.616578977482995,-0.651386560588766,0.321132992047611,-0.30397288469354],[0,0,0,0],[8.999999E+09,8.999999E+09,8.999999E+09,8.999999E+09,8.999999E+09,8.999999E+09]];
	LOCAL CONST Robtarget Tr_meulage_bavure_P442 :=[[68.9675625,-251.49840625,18.5],[0.621194857997989,-0.643210262813619,0.322004582054159,-0.31098320749555],[0,0,0,0],[8.999999E+09,8.999999E+09,8.999999E+09,8.999999E+09,8.999999E+09,8.999999E+09]];
	LOCAL CONST Robtarget Tr_meulage_bavure_P443 :=[[67.536953125,-249.237015625,18.5],[0.625274064526456,-0.635118117478085,0.323163750874937,-0.318154854123114],[0,0,0,0],[8.999999E+09,8.999999E+09,8.999999E+09,8.999999E+09,8.999999E+09,8.999999E+09]];
	LOCAL CONST Robtarget Tr_meulage_bavure_P444 :=[[65.30841015625,-246.166375,18.5],[0.629195870654258,-0.627595801253755,0.323806074960061,-0.324631625722519],[0,0,0,0],[8.999999E+09,8.999999E+09,8.999999E+09,8.999999E+09,8.999999E+09,8.999999E+09]];
	LOCAL CONST Robtarget Tr_meulage_bavure_P445 :=[[65.1301875,-245.9544375,18.5],[0.633407517469485,-0.621185253324401,0.323090991075483,-0.329448037406973],[0,0,0,0],[8.999999E+09,8.999999E+09,8.999999E+09,8.999999E+09,8.999999E+09,8.999999E+09]];
	LOCAL CONST Robtarget Tr_meulage_bavure_P446 :=[[63.8427421875,-243.8951875,18.5],[0.638324929987837,-0.61632361457984,0.320335376444725,-0.331770602171561],[0,0,0,0],[8.999999E+09,8.999999E+09,8.999999E+09,8.999999E+09,8.999999E+09,8.999999E+09]];
	LOCAL CONST Robtarget Tr_meulage_bavure_P447 :=[[63.10174609375,-242.643734375,18.5],[0.644197617322812,-0.613283286191339,0.315141437991395,-0.331027060487024],[0,0,0,0],[8.999999E+09,8.999999E+09,8.999999E+09,8.999999E+09,8.999999E+09,8.999999E+09]];
	LOCAL CONST Robtarget Tr_meulage_bavure_P448 :=[[62.6995859375,-242.080109375,18.5],[0.651033547744534,-0.612075038442941,0.307490006193705,-0.327061711481538],[0,0,0,0],[8.999999E+09,8.999999E+09,8.999999E+09,8.999999E+09,8.999999E+09,8.999999E+09]];
	LOCAL CONST Robtarget Tr_meulage_bavure_P449 :=[[61.8825390625,-240.82246875,18.5],[0.658553427410002,-0.612427778507783,0.297806281869182,-0.320235878436214],[0,0,0,0],[8.999999E+09,8.999999E+09,8.999999E+09,8.999999E+09,8.999999E+09,8.999999E+09]];
	LOCAL CONST Robtarget Tr_meulage_bavure_P450 :=[[60.37966796875,-238.573625,18.5],[0.666165976155559,-0.613794648518219,0.287068209026089,-0.311561976225696],[0,0,0,0],[8.999999E+09,8.999999E+09,8.999999E+09,8.999999E+09,8.999999E+09,8.999999E+09]];
	LOCAL CONST Robtarget Tr_meulage_bavure_P451 :=[[59.7568984375,-237.850484375,18.5],[0.673069205738495,-0.615442063047119,0.276760778527026,-0.302675375258663],[0,0,0,0],[8.999999E+09,8.999999E+09,8.999999E+09,8.999999E+09,8.999999E+09,8.999999E+09]];
	LOCAL CONST Robtarget Tr_meulage_bavure_P452 :=[[58.25674609375,-235.894515625,18.5],[0.678443486178576,-0.616627613312013,0.268602387613301,-0.295529321610267],[0,0,0,0],[8.999999E+09,8.999999E+09,8.999999E+09,8.999999E+09,8.999999E+09,8.999999E+09]];
	LOCAL CONST Robtarget Tr_meulage_bavure_P453 :=[[57.395265625,-234.48975,18.5],[0.681678889059586,-0.616783904091937,0.264052693884573,-0.291835026540505],[0,0,0,0],[8.999999E+09,8.999999E+09,8.999999E+09,8.999999E+09,8.999999E+09,8.999999E+09]];
	LOCAL CONST Robtarget Tr_meulage_bavure_P454 :=[[56.66391015625,-233.9003125,18.5],[0.682553555302259,-0.615627182985552,0.263791315207456,-0.292468729498797],[0,0,0,0],[8.999999E+09,8.999999E+09,8.999999E+09,8.999999E+09,8.999999E+09,8.999999E+09]];
	LOCAL CONST Robtarget Tr_meulage_bavure_P455 :=[[56.1930234375,-233.3075,18.5],[0.681220519414288,-0.613239367478987,0.267516208767153,-0.297171937015844],[0,0,0,0],[8.999999E+09,8.999999E+09,8.999999E+09,8.999999E+09,8.999999E+09,8.999999E+09]];
	LOCAL CONST Robtarget Tr_meulage_bavure_P456 :=[[54.596953125,-230.847265625,18.5],[0.678195680714665,-0.609995373743467,0.274063730134188,-0.304705324036971],[0,0,0,0],[8.999999E+09,8.999999E+09,8.999999E+09,8.999999E+09,8.999999E+09,8.999999E+09]];
	LOCAL CONST Robtarget Tr_meulage_bavure_P457 :=[[53.770875,-229.72215625,18.5],[0.674240624483602,-0.60646810737329,0.281826594421193,-0.313320579777285],[0,0,0,0],[8.999999E+09,8.999999E+09,8.999999E+09,8.999999E+09,8.999999E+09,8.999999E+09]];
	LOCAL CONST Robtarget Tr_meulage_bavure_P458 :=[[52.55294921875,-227.842796875,18.5],[0.670133470315653,-0.603246536344281,0.289328644273148,-0.321408904597229],[0,0,0,0],[8.999999E+09,8.999999E+09,8.999999E+09,8.999999E+09,8.999999E+09,8.999999E+09]];
	LOCAL CONST Robtarget Tr_meulage_bavure_P459 :=[[52.28729296875,-227.2823125,18.5],[0.666468975408144,-0.600719564184368,0.295616750605547,-0.327972326250217],[0,0,0,0],[8.999999E+09,8.999999E+09,8.999999E+09,8.999999E+09,8.999999E+09,8.999999E+09]];
	LOCAL CONST Robtarget Tr_meulage_bavure_P460 :=[[50.443359375,-225.00878125,18.5],[0.663476290719761,-0.599040042289513,0.300409183193492,-0.332722950875867],[0,0,0,0],[8.999999E+09,8.999999E+09,8.999999E+09,8.999999E+09,8.999999E+09,8.999999E+09]];
	LOCAL CONST Robtarget Tr_meulage_bavure_P461 :=[[49.62457421875,-224.007921875,18.5],[0.661098528492342,-0.598066265492912,0.30394585427408,-0.335979754411216],[0,0,0,0],[8.999999E+09,8.999999E+09,8.999999E+09,8.999999E+09,8.999999E+09,8.999999E+09]];
	LOCAL CONST Robtarget Tr_meulage_bavure_P462 :=[[48.3818359375,-222.254515625,18.5],[0.659097226720856,-0.597511432559076,0.306737669661884,-0.338353270562697],[0,0,0,0],[8.999999E+09,8.999999E+09,8.999999E+09,8.999999E+09,8.999999E+09,8.999999E+09]];
	LOCAL CONST Robtarget Tr_meulage_bavure_P463 :=[[47.44912890625,-220.926640625,18.5],[0.657160434538022,-0.597067593660473,0.309366788251912,-0.340503512764534],[0,0,0,0],[8.999999E+09,8.999999E+09,8.999999E+09,8.999999E+09,8.999999E+09,8.999999E+09]];
	LOCAL CONST Robtarget Tr_meulage_bavure_P464 :=[[46.1441328125,-218.79271875,18.5],[0.655058859189659,-0.596483867701833,0.312261202601386,-0.34292539701594],[0,0,0,0],[8.999999E+09,8.999999E+09,8.999999E+09,8.999999E+09,8.999999E+09,8.999999E+09]];
	LOCAL CONST Robtarget Tr_meulage_bavure_P465 :=[[44.40310546875,-216.575953125,18.5],[0.652668108638846,-0.595631591414993,0.31563718646446,-0.345861986629107],[0,0,0,0],[8.999999E+09,8.999999E+09,8.999999E+09,8.999999E+09,8.999999E+09,8.999999E+09]];
	LOCAL CONST Robtarget Tr_meulage_bavure_P466 :=[[43.8765859375,-215.836453125,18.5],[0.649967666943387,-0.594501718154504,0.319509171252316,-0.349318806429272],[0,0,0,0],[8.999999E+09,8.999999E+09,8.999999E+09,8.999999E+09,8.999999E+09,8.999999E+09]];
	LOCAL CONST Robtarget Tr_meulage_bavure_P467 :=[[42.58715625,-213.990453125,18.5],[0.647044365227752,-0.593183112516432,0.323708235105574,-0.353101066236238],[0,0,0,0],[8.999999E+09,8.999999E+09,8.999999E+09,8.999999E+09,8.999999E+09,8.999999E+09]];
	LOCAL CONST Robtarget Tr_meulage_bavure_P468 :=[[41.81332421875,-212.7619375,18.5],[0.644026093350293,-0.591828032106892,0.327991412268912,-0.356919605757778],[0,0,0,0],[8.999999E+09,8.999999E+09,8.999999E+09,8.999999E+09,8.999999E+09,8.999999E+09]];
	LOCAL CONST Robtarget Tr_meulage_bavure_P469 :=[[41.294921875,-212.04809375,18.5],[0.641082066659871,-0.590592668576113,0.332079193078546,-0.360468435727119],[0,0,0,0],[8.999999E+09,8.999999E+09,8.999999E+09,8.999999E+09,8.999999E+09,8.999999E+09]];
	LOCAL CONST Robtarget Tr_meulage_bavure_P470 :=[[39.0729375,-208.482265625,18.5],[0.638368318744693,-0.589660244068546,0.335707408568728,-0.363438058023876],[0,0,0,0],[8.999999E+09,8.999999E+09,8.999999E+09,8.999999E+09,8.999999E+09,8.999999E+09]];
	LOCAL CONST Robtarget Tr_meulage_bavure_P471 :=[[38.05090234375,-207.2359375,18.5],[0.636039593889692,-0.5891988162971,0.338630504075899,-0.365551325518093],[0,0,0,0],[8.999999E+09,8.999999E+09,8.999999E+09,8.999999E+09,8.999999E+09,8.999999E+09]];
	LOCAL CONST Robtarget Tr_meulage_bavure_P472 :=[[37.65609765625,-206.725765625,18.5],[0.634234388742189,-0.589349306026773,0.3406367517771,-0.366579785260084],[0,0,0,0],[8.999999E+09,8.999999E+09,8.999999E+09,8.999999E+09,8.999999E+09,8.999999E+09]];
	LOCAL CONST Robtarget Tr_meulage_bavure_P473 :=[[36.66534375,-205.104328125,18.5],[0.633027144384228,-0.590220326167077,0.341596784146684,-0.36637172122398],[0,0,0,0],[8.999999E+09,8.999999E+09,8.999999E+09,8.999999E+09,8.999999E+09,8.999999E+09]];
	LOCAL CONST Robtarget Tr_meulage_bavure_P474 :=[[36.46398828125,-204.721828125,18.5],[0.632450290569136,-0.591817871068681,0.341465921999909,-0.364909936224684],[0,0,0,0],[8.999999E+09,8.999999E+09,8.999999E+09,8.999999E+09,8.999999E+09,8.999999E+09]];
	LOCAL CONST Robtarget Tr_meulage_bavure_P475 :=[[35.49823046875,-203.681625,18.5],[0.632422261565449,-0.59407143673851,0.340354230218391,-0.362326108775411],[0,0,0,0],[8.999999E+09,8.999999E+09,8.999999E+09,8.999999E+09,8.999999E+09,8.999999E+09]];
	LOCAL CONST Robtarget Tr_meulage_bavure_P476 :=[[35.11794921875,-203.1165,18.5],[0.632782105568893,-0.596819668869092,0.338502669162777,-0.358899752984675],[0,0,0,0],[8.999999E+09,8.999999E+09,8.999999E+09,8.999999E+09,8.999999E+09,8.999999E+09]];
	LOCAL CONST Robtarget Tr_meulage_bavure_P477 :=[[29.08728125,-194.351140625,18.5],[0.633334711106061,-0.599840860684526,0.336229554403492,-0.355003904636383],[0,0,0,0],[8.999999E+09,8.999999E+09,8.999999E+09,8.999999E+09,8.999999E+09,8.999999E+09]];
	LOCAL CONST Robtarget Tr_meulage_bavure_P478 :=[[29.06719921875,-194.320421875,18.5],[0.633876454034294,-0.602918627091504,0.333877399375168,-0.351020871620878],[0,0,0,0],[8.999999E+09,8.999999E+09,8.999999E+09,8.999999E+09,8.999999E+09,8.999999E+09]];
	LOCAL CONST Robtarget Tr_meulage_bavure_P479 :=[[29.047515625,-194.293734375,18.5],[0.634259217791597,-0.60586565243574,0.331727412566561,-0.347273637923902],[0,0,0,0],[8.999999E+09,8.999999E+09,8.999999E+09,8.999999E+09,8.999999E+09,8.999999E+09]];
	LOCAL CONST Robtarget Tr_meulage_bavure_P480 :=[[26.49462890625,-190.371140625,18.5],[0.634379112746677,-0.608558519584429,0.329987340406716,-0.34398840783266],[0,0,0,0],[8.999999E+09,8.999999E+09,8.999999E+09,8.999999E+09,8.999999E+09,8.999999E+09]];
	LOCAL CONST Robtarget Tr_meulage_bavure_P481 :=[[25.48696875,-189.150890625,18.5],[0.634199561362685,-0.610914546722038,0.328768681131607,-0.341299703014474],[0,0,0,0],[8.999999E+09,8.999999E+09,8.999999E+09,8.999999E+09,8.999999E+09,8.999999E+09]];
	LOCAL CONST Robtarget Tr_meulage_bavure_P482 :=[[24.021576171875,-187.23075,18.5],[0.633731228605643,-0.612886416916352,0.328106414293023,-0.339265605019419],[0,0,0,0],[8.999999E+09,8.999999E+09,8.999999E+09,8.999999E+09,8.999999E+09,8.999999E+09]];
	LOCAL CONST Robtarget Tr_meulage_bavure_P483 :=[[23.547546875,-186.559203125,18.5],[0.633014866821095,-0.614493939254942,0.327954478711378,-0.337839069522108],[0,0,0,0],[8.999999E+09,8.999999E+09,8.999999E+09,8.999999E+09,8.999999E+09,8.999999E+09]];
	LOCAL CONST Robtarget Tr_meulage_bavure_P484 :=[[23.32076953125,-186.219703125,18.5],[0.632158365379361,-0.615830031919444,0.328133949714492,-0.336834208345527],[0,0,0,0],[8.999999E+09,8.999999E+09,8.999999E+09,8.999999E+09,8.999999E+09,8.999999E+09]];
	LOCAL CONST Robtarget Tr_meulage_bavure_P485 :=[[22.992279296875,-185.695,18.5],[0.631341909765972,-0.617043790856116,0.328336985475419,-0.335945199560707],[0,0,0,0],[8.999999E+09,8.999999E+09,8.999999E+09,8.999999E+09,8.999999E+09,8.999999E+09]];
	LOCAL CONST Robtarget Tr_meulage_bavure_P486 :=[[20.67498828125,-181.834375,18.5],[0.630764108757581,-0.618319336608578,0.328205825266584,-0.334811548994748],[0,0,0,0],[8.999999E+09,8.999999E+09,8.999999E+09,8.999999E+09,8.999999E+09,8.999999E+09]];
	LOCAL CONST Robtarget Tr_meulage_bavure_P487 :=[[19.530822265625,-180.427234375,18.5],[0.630578338165765,-0.619793385173804,0.327462064933538,-0.333160194441596],[0,0,0,0],[8.999999E+09,8.999999E+09,8.999999E+09,8.999999E+09,8.999999E+09,8.999999E+09]];
	LOCAL CONST Robtarget Tr_meulage_bavure_P488 :=[[17.601287109375,-177.76746875,18.5],[0.630795360347721,-0.621495583118767,0.326063549523254,-0.330942616173787],[0,0,0,0],[8.999999E+09,8.999999E+09,8.999999E+09,8.999999E+09,8.999999E+09,8.999999E+09]];
	LOCAL CONST Robtarget Tr_meulage_bavure_P489 :=[[15.6425478515625,-175.167546875,18.5],[0.631290643631171,-0.623301956071415,0.324233518597492,-0.328389129295077],[0,0,0,0],[8.999999E+09,8.999999E+09,8.999999E+09,8.999999E+09,8.999999E+09,8.999999E+09]];
	LOCAL CONST Robtarget Tr_meulage_bavure_P490 :=[[13.9278564453125,-172.6341875,18.5],[0.631843505848642,-0.624997668994709,0.322383647530065,-0.32591483806861],[0,0,0,0],[8.999999E+09,8.999999E+09,8.999999E+09,8.999999E+09,8.999999E+09,8.999999E+09]];
	LOCAL CONST Robtarget Tr_meulage_bavure_P491 :=[[12.678619140625,-170.9785,18.5],[0.632235623072412,-0.626367269395334,0.320938548140575,-0.323945379756977],[0,0,0,0],[8.999999E+09,8.999999E+09,8.999999E+09,8.999999E+09,8.999999E+09,8.999999E+09]];
	LOCAL CONST Robtarget Tr_meulage_bavure_P492 :=[[11.3559267578125,-169.02978125,18.5],[0.632349816479591,-0.627274718884118,0.320152208501845,-0.322742467051471],[0,0,0,0],[8.999999E+09,8.999999E+09,8.999999E+09,8.999999E+09,8.999999E+09,8.999999E+09]];
	LOCAL CONST Robtarget Tr_meulage_bavure_P493 :=[[11.05386328125,-168.457984375,18.5],[0.632170540851071,-0.627721043692541,0.32005418998209,-0.322322841357109],[0,0,0,0],[8.999999E+09,8.999999E+09,8.999999E+09,8.999999E+09,8.999999E+09,8.999999E+09]];
	LOCAL CONST Robtarget Tr_meulage_bavure_P494 :=[[9.4859921875,-166.529390625,18.5],[0.631806376119159,-0.627788398439396,0.320455710159719,-0.322506694048518],[0,0,0,0],[8.999999E+09,8.999999E+09,8.999999E+09,8.999999E+09,8.999999E+09,8.999999E+09]];
	LOCAL CONST Robtarget Tr_meulage_bavure_P495 :=[[8.354400390625,-164.83940625,18.5],[0.631395404318594,-0.627610824370775,0.321089823190818,-0.323026039169112],[0,0,0,0],[8.999999E+09,8.999999E+09,8.999999E+09,8.999999E+09,8.999999E+09,8.999999E+09]];
	LOCAL CONST Robtarget Tr_meulage_bavure_P496 :=[[6.9548037109375,-162.967875,18.5],[0.631062583044117,-0.627292606713559,0.321726680291029,-0.323660230848815],[0,0,0,0],[8.999999E+09,8.999999E+09,8.999999E+09,8.999999E+09,8.999999E+09,8.999999E+09]];
	LOCAL CONST Robtarget Tr_meulage_bavure_P497 :=[[5.6199951171875,-161.0065625,18.5],[0.630877249951225,-0.626884132427577,0.322244526788264,-0.324297155336756],[0,0,0,0],[8.999999E+09,8.999999E+09,8.999999E+09,8.999999E+09,8.999999E+09,8.999999E+09]];
	LOCAL CONST Robtarget Tr_meulage_bavure_P498 :=[[3.42715454101563,-157.928078125,18.5],[0.630850521804765,-0.626378331911445,0.322634545387148,-0.324938078059987],[0,0,0,0],[8.999999E+09,8.999999E+09,8.999999E+09,8.999999E+09,8.999999E+09,8.999999E+09]];
	LOCAL CONST Robtarget Tr_meulage_bavure_P499 :=[[2.83883666992188,-157.0609375,18.5],[0.630962129544759,-0.625734388814637,0.322949902571821,-0.325648009611553],[0,0,0,0],[8.999999E+09,8.999999E+09,8.999999E+09,8.999999E+09,8.999999E+09,8.999999E+09]];
	LOCAL CONST Robtarget Tr_meulage_bavure_P500 :=[[1.487060546875,-155.26353125,18.5],[0.631172232372544,-0.624920783688008,0.323260325283402,-0.326494087686582],[0,0,0,0],[8.999999E+09,8.999999E+09,8.999999E+09,8.999999E+09,8.999999E+09,8.999999E+09]];
	LOCAL CONST Robtarget Tr_meulage_bavure_P501 :=[[0.62982177734375,-153.96803125,18.5],[0.631457344562057,-0.623913923941822,0.323608894150449,-0.327521481947181],[0,0,0,0],[8.999999E+09,8.999999E+09,8.999999E+09,8.999999E+09,8.999999E+09,8.999999E+09]];
	LOCAL CONST Robtarget Tr_meulage_bavure_P502 :=[[0.2587890625,-153.4425,18.5],[0.631819374844419,-0.622707697724944,0.323994550654934,-0.328735352390359],[0,0,0,0],[8.999999E+09,8.999999E+09,8.999999E+09,8.999999E+09,8.999999E+09,8.999999E+09]];
	LOCAL CONST Robtarget Tr_meulage_bavure_P503 :=[[-1.5235595703125,-150.646,18.5],[0.632267055268863,-0.621342153073936,0.324376065041991,-0.330079487491968],[0,0,0,0],[8.999999E+09,8.999999E+09,8.999999E+09,8.999999E+09,8.999999E+09,8.999999E+09]];
	LOCAL CONST Robtarget Tr_meulage_bavure_P504 :=[[-2.75897216796875,-149.140328125,18.5],[0.632835495809181,-0.619869173804311,0.324673150523223,-0.331464610389154],[0,0,0,0],[8.999999E+09,8.999999E+09,8.999999E+09,8.999999E+09,8.999999E+09,8.999999E+09]];
	LOCAL CONST Robtarget Tr_meulage_bavure_P505 :=[[-3.681884765625,-147.7770625,18.5],[0.633587340054045,-0.618387042583769,0.324743273775202,-0.332725644075572],[0,0,0,0],[8.999999E+09,8.999999E+09,8.999999E+09,8.999999E+09,8.999999E+09,8.999999E+09]];
	LOCAL CONST Robtarget Tr_meulage_bavure_P506 :=[[-5.831939453125,-144.632359375,18.5],[0.634618975220367,-0.617043055691565,0.324374121562303,-0.333613628279407],[0,0,0,0],[8.999999E+09,8.999999E+09,8.999999E+09,8.999999E+09,8.999999E+09,8.999999E+09]];
	LOCAL CONST Robtarget Tr_meulage_bavure_P507 :=[[-5.8612978515625,-144.573625,18.5],[0.636059947260741,-0.615975877111349,0.323321380123199,-0.333863366458191],[0,0,0,0],[8.999999E+09,8.999999E+09,8.999999E+09,8.999999E+09,8.999999E+09,8.999999E+09]];
	LOCAL CONST Robtarget Tr_meulage_bavure_P508 :=[[-6.0228271484375,-144.34259375,18.5],[0.63798375914842,-0.615312394507583,0.321414348105098,-0.333256953506406],[0,0,0,0],[8.999999E+09,8.999999E+09,8.999999E+09,8.999999E+09,8.999999E+09,8.999999E+09]];
	LOCAL CONST Robtarget Tr_meulage_bavure_P509 :=[[-8.08917236328125,-140.99503125,18.5],[0.640351779243819,-0.615051431796167,0.318695393147869,-0.331805035300981],[0,0,0,0],[8.999999E+09,8.999999E+09,8.999999E+09,8.999999E+09,8.999999E+09,8.999999E+09]];
	LOCAL CONST Robtarget Tr_meulage_bavure_P510 :=[[-9.461486328125,-139.18734375,18.5],[0.642943210041017,-0.615032860953445,0.315529375694305,-0.329848179748708],[0,0,0,0],[8.999999E+09,8.999999E+09,8.999999E+09,8.999999E+09,8.999999E+09,8.999999E+09]];
	LOCAL CONST Robtarget Tr_meulage_bavure_P511 :=[[-11.4542236328125,-136.315140625,18.5],[0.645393997720774,-0.614950490789474,0.312562105309861,-0.328035686942825],[0,0,0,0],[8.999999E+09,8.999999E+09,8.999999E+09,8.999999E+09,8.999999E+09,8.999999E+09]];
	LOCAL CONST Robtarget Tr_meulage_bavure_P512 :=[[-13.1698916015625,-134.277671875,18.5],[0.647311411625241,-0.614466358222711,0.310512392692234,-0.327110203107149],[0,0,0,0],[8.999999E+09,8.999999E+09,8.999999E+09,8.999999E+09,8.999999E+09,8.999999E+09]];
	LOCAL CONST Robtarget Tr_meulage_bavure_P513 :=[[-14.68051171875,-132.192265625,18.5],[0.64843152158747,-0.613374264794576,0.309854868809359,-0.327564548409328],[0,0,0,0],[8.999999E+09,8.999999E+09,8.999999E+09,8.999999E+09,8.999999E+09,8.999999E+09]];
	LOCAL CONST Robtarget Tr_meulage_bavure_P514 :=[[-15.8515625,-130.537875,18.5],[0.648742592834258,-0.611703732914464,0.310577501507567,-0.329383070206274],[0,0,0,0],[8.999999E+09,8.999999E+09,8.999999E+09,8.999999E+09,8.999999E+09,8.999999E+09]];
	LOCAL CONST Robtarget Tr_meulage_bavure_P515 :=[[-20.22738671875,-124.304578125,18.5],[0.648518889569445,-0.609725142451844,0.312142395640959,-0.332002447848227],[0,0,0,0],[8.999999E+09,8.999999E+09,8.999999E+09,8.999999E+09,8.999999E+09,8.999999E+09]];
	LOCAL CONST Robtarget Tr_meulage_bavure_P516 :=[[-20.891326171875,-123.3272109375,18.5],[0.64819817785806,-0.607881098388929,0.313713316860279,-0.33452002521147],[0,0,0,0],[8.999999E+09,8.999999E+09,8.999999E+09,8.999999E+09,8.999999E+09,8.999999E+09]];
	LOCAL CONST Robtarget Tr_meulage_bavure_P517 :=[[-21.53335546875,-122.3264140625,18.5],[0.648230450450731,-0.606581954602119,0.314489813791291,-0.33608298451578],[0,0,0,0],[8.999999E+09,8.999999E+09,8.999999E+09,8.999999E+09,8.999999E+09,8.999999E+09]];
	LOCAL CONST Robtarget Tr_meulage_bavure_P518 :=[[-21.969359375,-121.736890625,18.5],[0.648882644235928,-0.60606323345056,0.314016735937517,-0.336202558913506],[0,0,0,0],[8.999999E+09,8.999999E+09,8.999999E+09,8.999999E+09,8.999999E+09,8.999999E+09]];
	LOCAL CONST Robtarget Tr_meulage_bavure_P519 :=[[-23.89407421875,-118.7724140625,18.5],[0.650151172006559,-0.60631224444472,0.312309388098864,-0.334890671533586],[0,0,0,0],[8.999999E+09,8.999999E+09,8.999999E+09,8.999999E+09,8.999999E+09,8.999999E+09]];
	LOCAL CONST Robtarget Tr_meulage_bavure_P520 :=[[-27.6311953125,-113.9946171875,18.5],[0.65179619183045,-0.607088644818988,0.309797514143522,-0.332611788542832],[0,0,0,0],[8.999999E+09,8.999999E+09,8.999999E+09,8.999999E+09,8.999999E+09,8.999999E+09]];
	LOCAL CONST Robtarget Tr_meulage_bavure_P521 :=[[-28.2760625,-113.084546875,18.5],[0.653461561430621,-0.608044595604171,0.307125704709975,-0.330065991879829],[0,0,0,0],[8.999999E+09,8.999999E+09,8.999999E+09,8.999999E+09,8.999999E+09,8.999999E+09]];
	LOCAL CONST Robtarget Tr_meulage_bavure_P522 :=[[-28.87939453125,-112.25334375,18.5],[0.654806667164718,-0.608836043695375,0.304938203258267,-0.327962791681644],[0,0,0,0],[8.999999E+09,8.999999E+09,8.999999E+09,8.999999E+09,8.999999E+09,8.999999E+09]];
	LOCAL CONST Robtarget Tr_meulage_bavure_P523 :=[[-30.689361328125,-109.5281796875,18.5],[0.655624756804297,-0.609246102660619,0.303647337826473,-0.326762389036817],[0,0,0,0],[8.999999E+09,8.999999E+09,8.999999E+09,8.999999E+09,8.999999E+09,8.999999E+09]];
	LOCAL CONST Robtarget Tr_meulage_bavure_P524 :=[[-31.3649296875,-108.601640625,18.5],[0.655888538248224,-0.609250742454429,0.303314682189269,-0.326533247590132],[0,0,0,0],[8.999999E+09,8.999999E+09,8.999999E+09,8.999999E+09,8.999999E+09,8.999999E+09]];
	LOCAL CONST Robtarget Tr_meulage_bavure_P525 :=[[-31.945587890625,-107.7489140625,18.5],[0.655766631435243,-0.608972696053468,0.303651045057075,-0.326983827418407],[0,0,0,0],[8.999999E+09,8.999999E+09,8.999999E+09,8.999999E+09,8.999999E+09,8.999999E+09]];
	LOCAL CONST Robtarget Tr_meulage_bavure_P526 :=[[-32.83975390625,-106.2560546875,18.5],[0.655521281122365,-0.608663407179975,0.304161179589592,-0.327576988792598],[0,0,0,0],[8.999999E+09,8.999999E+09,8.999999E+09,8.999999E+09,8.999999E+09,8.999999E+09]];
	LOCAL CONST Robtarget Tr_meulage_bavure_P527 :=[[-34.50521875,-104.0425546875,18.5],[0.655407258002898,-0.608530495729236,0.304390715907491,-0.327838762189553],[0,0,0,0],[8.999999E+09,8.999999E+09,8.999999E+09,8.999999E+09,8.999999E+09,8.999999E+09]];
	LOCAL CONST Robtarget Tr_meulage_bavure_degg1 :=[[-42.4852141289787,-110.023439249339,17.7592614432629],[0.655407258002898,-0.608530495729236,0.304390715907491,-0.327838762189553],[0,0,0,0],[8.999999E+09,8.999999E+09,8.999999E+09,8.999999E+09,8.999999E+09,8.999999E+09]];
	LOCAL CONST Robtarget Tr_meulage_bavure_degg2 :=[[-194.105126329574,-223.660245924276,3.68522886525799],[0.655407258002898,-0.608530495729236,0.304390715907491,-0.327838762189553],[0,0,0,0],[8.999999E+09,8.999999E+09,8.999999E+09,8.999999E+09,8.999999E+09,8.999999E+09]];
	LOCAL PROC Tr_pick()
		!!Programme Tr_pick - 28/02/2023 14:40:20;
		 CONST Robtarget Ppick :=[[-47.6699981689453,-10.8400001525879,634.599975585938],[0.00986171453897316,-0.924580919553334,0.379718018337624,-0.0294464995204969],[0,0,0,0],[8.999999E+09,8.999999E+09,8.999999E+09,8.999999E+09,8.999999E+09,8.999999E+09]];
		 VAR Pose Ref :=[[0,0,0],[1,0,0,0]];
		LocalisationPieceTable 6 \model:=0;
		MoveJ Reltool(Ppick,0,0,-200),V1000,Z0,Tool_Prehenseur \Wobj:=Wobj_vision;
		MoveL Reltool(Ppick,0,0,-100),V500,Z0,Tool_Prehenseur \Wobj:=Wobj_vision;
		MoveL Reltool(Ppick,0,0,-10),V200,Z0,Tool_Prehenseur \Wobj:=Wobj_vision;
		MoveL Ppick,V100,Fine,Tool_Prehenseur \Wobj:=Wobj_vision;
		Gripper_Close;
		MoveL Reltool(Ppick,0,0,-200),V500,Z0,Tool_Prehenseur \Wobj:=Wobj_vision;
		LocalisationPiecePrehenseur 6 \model:=0,Ref;
	ENDPROC
	LOCAL PROC Tr_Cut()
		!!Programme Tr_Cut - 28/02/2023 14:40:20;
		confJ \off;
		confL \off;
		Tool := ToolOffset(Tool_M2_D490_S180);
		MoveAbsJ [[0,-40,40,0,90,0],[8.999999E+09,8.999999E+09,8.999999E+09,8.999999E+09,8.999999E+09,8.999999E+09]] ,V1000,Z0,Tool_M2_D490_S180 \Wobj:=Wobj_Part_0;
		Movej Reltool(Coupe_0,-200,0,-45.08496484375),V1000,Z0,Tool_M2_D490_S180 \Wobj:=Wobj_Part_0;
		MoveL Reltool(Coupe_0,0,0,-45.08496484375),V500,Z0,Tool_M2_D490_S180 \Wobj:=Wobj_Part_0;
		MoveL Reltool(Coupe_0,0,0,-35.08496484375),vitesse_Tronconnage,Z0,Tool_M2_D490_S180 \Wobj:=Wobj_Part_0;
		MoveL Coupe_0,vitesse_Tronconnage,Fine,Tool_M2_D490_S180 \Wobj:=Wobj_Part_0;
		MoveL Reltool(Coupe_0,0,0,35.08496484375),vitesse_Tronconnage,Z0,Tool_M2_D490_S180 \Wobj:=Wobj_Part_0;
